//     PlcTask Inputs/GVL_iXlinker.EtherCAT_Master_BKCUCX.Beckhoff_CUxxxx.Beckhoff_CUxxxxEK1122.A_0001_CU1123_0000_0016.A_0002_CU1123_0010_0016.A_0003_CU1124_0000_0016.A_0004_CU1128_0000_0000.A_0005_CU1128_0000_0001.A_0006_CU1128_0000_0002.A_0013_CU2508_0000_0019.EPM_Inputs_Channel_1.Dropped_frames_tx <-> EPM Inputs Channel 1/Dropped frames tx
//     PlcTask Inputs/GVL_iXlinker.EtherCAT_Master_BKCUCX.Beckhoff_CUxxxx.Beckhoff_CUxxxxEK1122.A_0001_CU1123_0000_0016.A_0002_CU1123_0010_0016.A_0003_CU1124_0000_0016.A_0004_CU1128_0000_0000.A_0005_CU1128_0000_0001.A_0006_CU1128_0000_0002.A_0013_CU2508_0000_0019.EPM_Inputs_Channel_2.Dropped_frames_tx <-> EPM Inputs Channel 2/Dropped frames tx
//     PlcTask Inputs/GVL_iXlinker.EtherCAT_Master_BKCUCX.Beckhoff_CUxxxx.Beckhoff_CUxxxxEK1122.A_0001_CU1123_0000_0016.A_0002_CU1123_0010_0016.A_0003_CU1124_0000_0016.A_0004_CU1128_0000_0000.A_0005_CU1128_0000_0001.A_0006_CU1128_0000_0002.A_0013_CU2508_0000_0019.EPM_Inputs_Channel_3.Dropped_frames_tx <-> EPM Inputs Channel 3/Dropped frames tx
//     PlcTask Inputs/GVL_iXlinker.EtherCAT_Master_BKCUCX.Beckhoff_CUxxxx.Beckhoff_CUxxxxEK1122.A_0001_CU1123_0000_0016.A_0002_CU1123_0010_0016.A_0003_CU1124_0000_0016.A_0004_CU1128_0000_0000.A_0005_CU1128_0000_0001.A_0006_CU1128_0000_0002.A_0013_CU2508_0000_0019.EPM_Inputs_Channel_4.Dropped_frames_tx <-> EPM Inputs Channel 4/Dropped frames tx
//     PlcTask Inputs/GVL_iXlinker.EtherCAT_Master_BKCUCX.Beckhoff_CUxxxx.Beckhoff_CUxxxxEK1122.A_0001_CU1123_0000_0016.A_0002_CU1123_0010_0016.A_0003_CU1124_0000_0016.A_0004_CU1128_0000_0000.A_0005_CU1128_0000_0001.A_0006_CU1128_0000_0002.A_0013_CU2508_0000_0019.EPM_Inputs_Channel_5.Dropped_frames_tx <-> EPM Inputs Channel 5/Dropped frames tx
//     PlcTask Inputs/GVL_iXlinker.EtherCAT_Master_BKCUCX.Beckhoff_CUxxxx.Beckhoff_CUxxxxEK1122.A_0001_CU1123_0000_0016.A_0002_CU1123_0010_0016.A_0003_CU1124_0000_0016.A_0004_CU1128_0000_0000.A_0005_CU1128_0000_0001.A_0006_CU1128_0000_0002.A_0013_CU2508_0000_0019.EPM_Inputs_Channel_6.Dropped_frames_tx <-> EPM Inputs Channel 6/Dropped frames tx
//     PlcTask Inputs/GVL_iXlinker.EtherCAT_Master_BKCUCX.Beckhoff_CUxxxx.Beckhoff_CUxxxxEK1122.A_0001_CU1123_0000_0016.A_0002_CU1123_0010_0016.A_0003_CU1124_0000_0016.A_0004_CU1128_0000_0000.A_0005_CU1128_0000_0001.A_0006_CU1128_0000_0002.A_0013_CU2508_0000_0019.EPM_Inputs_Channel_7.Dropped_frames_tx <-> EPM Inputs Channel 7/Dropped frames tx
//     PlcTask Inputs/GVL_iXlinker.EtherCAT_Master_BKCUCX.Beckhoff_CUxxxx.Beckhoff_CUxxxxEK1122.A_0001_CU1123_0000_0016.A_0002_CU1123_0010_0016.A_0003_CU1124_0000_0016.A_0004_CU1128_0000_0000.A_0005_CU1128_0000_0001.A_0006_CU1128_0000_0002.A_0013_CU2508_0000_0019.EPM_Inputs_Channel_8.Dropped_frames_tx <-> EPM Inputs Channel 8/Dropped frames tx
//     PlcTask Inputs/GVL_iXlinker.EtherCAT_Master_BKCUCX.Beckhoff_CUxxxx.Beckhoff_CUxxxxEK1122.A_0001_CU1123_0000_0016.A_0002_CU1123_0010_0016.A_0003_CU1124_0000_0016.A_0004_CU1128_0000_0000.A_0005_CU1128_0000_0001.A_0006_CU1128_0000_0002.A_0013_CU2508_0000_0019.EPM_Inputs_Channel_9.Dropped_frames_tx <-> EPM Inputs Channel 9/Dropped frames tx
//     PlcTask Inputs/GVL_iXlinker.EtherCAT_Master_BKCUCX.Beckhoff_CUxxxx.Beckhoff_CUxxxxEK1122.A_0001_CU1123_0000_0016.A_0002_CU1123_0010_0016.A_0003_CU1124_0000_0016.A_0004_CU1128_0000_0000.A_0005_CU1128_0000_0001.A_0006_CU1128_0000_0002.A_0013_CU2508_0000_0019.EPM_Inputs_Channel_10.Dropped_frames_tx <-> EPM Inputs Channel 10/Dropped frames tx
//     PlcTask Inputs/GVL_iXlinker.EtherCAT_Master_BKCUCX.Beckhoff_CUxxxx.Beckhoff_CUxxxxEK1122.A_0001_CU1123_0000_0016.A_0002_CU1123_0010_0016.A_0003_CU1124_0000_0016.A_0004_CU1128_0000_0000.A_0005_CU1128_0000_0001.A_0006_CU1128_0000_0002.A_0013_CU2508_0000_0019.WcState.WcState <-> WcState/WcState
//     PlcTask Inputs/GVL_iXlinker.EtherCAT_Master_BKCUCX.Beckhoff_CUxxxx.Beckhoff_CUxxxxEK1122.A_0001_CU1123_0000_0016.A_0002_CU1123_0010_0016.A_0003_CU1124_0000_0016.A_0004_CU1128_0000_0000.A_0005_CU1128_0000_0001.A_0006_CU1128_0000_0002.A_0013_CU2508_0000_0019.WcState.InputToggle <-> WcState/InputToggle
//     PlcTask Inputs/GVL_iXlinker.EtherCAT_Master_BKCUCX.Beckhoff_CUxxxx.Beckhoff_CUxxxxEK1122.A_0001_CU1123_0000_0016.A_0002_CU1123_0010_0016.A_0003_CU1124_0000_0016.A_0004_CU1128_0000_0000.A_0005_CU1128_0000_0001.A_0006_CU1128_0000_0002.A_0013_CU2508_0000_0019.InfoData.AdsAddr <-> InfoData/AdsAddr
//     PlcTask Inputs/GVL_iXlinker.EtherCAT_Master_BKCUCX.Beckhoff_CUxxxx.Beckhoff_CUxxxxEK1122.A_0001_CU1123_0000_0016.A_0002_CU1123_0010_0016.A_0003_CU1124_0000_0016.A_0004_CU1128_0000_0000.A_0005_CU1128_0000_0001.A_0006_CU1128_0000_0002.A_0013_CU2508_0000_0019.InfoData.State <-> InfoData/State
//   PLC/PLC Instance <-> EtherCAT Master BKCUCX/Beckhoff CUxxxx/Beckhoff CUxxxxEK1122/A_0001(CU1123-0000-0016)/A_0002(CU1123-0010-0016)/A_0003(CU1124-0000-0016)/A_0004(CU1128-0000-0000)/A_0005(CU1128-0000-0001)/A_0006(CU1128-0000-0002)/A_0006(CU1128-0000-0002)_2 (CU1128-B)
//     PlcTask Inputs/GVL_iXlinker.EtherCAT_Master_BKCUCX.Beckhoff_CUxxxx.Beckhoff_CUxxxxEK1122.A_0001_CU1123_0000_0016.A_0002_CU1123_0010_0016.A_0003_CU1124_0000_0016.A_0004_CU1128_0000_0000.A_0005_CU1128_0000_0001.A_0006_CU1128_0000_0002.A_0006_CU1128_0000_0002_2_CU1128_B.InfoData.State <-> InfoData/State
//   PLC/PLC Instance <-> EtherCAT Master BKCUCX/Beckhoff CUxxxx/Beckhoff CUxxxxEK1122/A_0001(CU1123-0000-0016)/A_0002(CU1123-0010-0016)/A_0003(CU1124-0000-0016)/A_0004(CU1128-0000-0000)/A_0005(CU1128-0000-0001)/A_0006(CU1128-0000-0002)/A_0006(CU1128-0000-0002)_3 (CU1128-C)
//     PlcTask Inputs/GVL_iXlinker.EtherCAT_Master_BKCUCX.Beckhoff_CUxxxx.Beckhoff_CUxxxxEK1122.A_0001_CU1123_0000_0016.A_0002_CU1123_0010_0016.A_0003_CU1124_0000_0016.A_0004_CU1128_0000_0000.A_0005_CU1128_0000_0001.A_0006_CU1128_0000_0002.A_0006_CU1128_0000_0002_3_CU1128_C.InfoData.State <-> InfoData/State
//   PLC/PLC Instance <-> EtherCAT Master BKCUCX/Beckhoff CUxxxx/Beckhoff CUxxxxEK1122/A_0001(CU1123-0000-0016)/A_0002(CU1123-0010-0016)/A_0003(CU1124-0000-0016)/A_0004(CU1128-0000-0000)/A_0005(CU1128-0000-0001)/A_0005(CU1128-0000-0001)_2 (CU1128-B)
//     PlcTask Inputs/GVL_iXlinker.EtherCAT_Master_BKCUCX.Beckhoff_CUxxxx.Beckhoff_CUxxxxEK1122.A_0001_CU1123_0000_0016.A_0002_CU1123_0010_0016.A_0003_CU1124_0000_0016.A_0004_CU1128_0000_0000.A_0005_CU1128_0000_0001.A_0005_CU1128_0000_0001_2_CU1128_B.InfoData.State <-> InfoData/State
//   PLC/PLC Instance <-> EtherCAT Master BKCUCX/Beckhoff CUxxxx/Beckhoff CUxxxxEK1122/A_0001(CU1123-0000-0016)/A_0002(CU1123-0010-0016)/A_0003(CU1124-0000-0016)/A_0004(CU1128-0000-0000)/A_0005(CU1128-0000-0001)/A_0005(CU1128-0000-0001)_3 (CU1128-C)
//     PlcTask Inputs/GVL_iXlinker.EtherCAT_Master_BKCUCX.Beckhoff_CUxxxx.Beckhoff_CUxxxxEK1122.A_0001_CU1123_0000_0016.A_0002_CU1123_0010_0016.A_0003_CU1124_0000_0016.A_0004_CU1128_0000_0000.A_0005_CU1128_0000_0001.A_0005_CU1128_0000_0001_3_CU1128_C.InfoData.State <-> InfoData/State
//   PLC/PLC Instance <-> EtherCAT Master BKCUCX/Beckhoff CUxxxx/Beckhoff CUxxxxEK1122/A_0001(CU1123-0000-0016)/A_0002(CU1123-0010-0016)/A_0003(CU1124-0000-0016)/A_0004(CU1128-0000-0000)/A_0004(CU1128-0000-0000)_2 (CU1128-B)
//     PlcTask Inputs/GVL_iXlinker.EtherCAT_Master_BKCUCX.Beckhoff_CUxxxx.Beckhoff_CUxxxxEK1122.A_0001_CU1123_0000_0016.A_0002_CU1123_0010_0016.A_0003_CU1124_0000_0016.A_0004_CU1128_0000_0000.A_0004_CU1128_0000_0000_2_CU1128_B.InfoData.State <-> InfoData/State
//   PLC/PLC Instance <-> EtherCAT Master BKCUCX/Beckhoff CUxxxx/Beckhoff CUxxxxEK1122/A_0001(CU1123-0000-0016)/A_0002(CU1123-0010-0016)/A_0003(CU1124-0000-0016)/A_0004(CU1128-0000-0000)/A_0004(CU1128-0000-0000)_3 (CU1128-C)
//     PlcTask Inputs/GVL_iXlinker.EtherCAT_Master_BKCUCX.Beckhoff_CUxxxx.Beckhoff_CUxxxxEK1122.A_0001_CU1123_0000_0016.A_0002_CU1123_0010_0016.A_0003_CU1124_0000_0016.A_0004_CU1128_0000_0000.A_0004_CU1128_0000_0000_3_CU1128_C.InfoData.State <-> InfoData/State
//   PLC/PLC Instance <-> EtherCAT Master BKCUCX/Beckhoff CXxxxx
//     PlcTask Inputs/GVL_iXlinker.EtherCAT_Master_BKCUCX.Beckhoff_CXxxxx.InfoData.State <-> InfoData/State
//   PLC/PLC Instance <-> EtherCAT Master BKCUCX/Beckhoff CXxxxx/Beckhoff CXxxxxEK1122
//     PlcTask Inputs/GVL_iXlinker.EtherCAT_Master_BKCUCX.Beckhoff_CXxxxx.Beckhoff_CXxxxxEK1122.InfoData.State <-> InfoData/State
//   PLC/PLC Instance <-> EtherCAT Master BKCUCX/Beckhoff CXxxxx/Beckhoff CXxxxxEK1122/Beckhoff CXxxxxsub EK1100
//     PlcTask Inputs/GVL_iXlinker.EtherCAT_Master_BKCUCX.Beckhoff_CXxxxx.Beckhoff_CXxxxxEK1122.Beckhoff_CXxxxxsub_EK1100.InfoData.State <-> InfoData/State
//   PLC/PLC Instance <-> EtherCAT Master BKCUCX/Beckhoff CXxxxx/Beckhoff CXxxxxEK1122/A_0001(CX1100-0004-0000)
//     PlcTask Inputs/GVL_iXlinker.EtherCAT_Master_BKCUCX.Beckhoff_CXxxxx.Beckhoff_CXxxxxEK1122.A_0001_CX1100_0004_0000.InfoData.State <-> InfoData/State
//   PLC/PLC Instance <-> EtherCAT Master BKCUCX/Beckhoff CXxxxx/Beckhoff CXxxxxEK1122/A_0003(CX1100-0004-0002)
//     PlcTask Inputs/GVL_iXlinker.EtherCAT_Master_BKCUCX.Beckhoff_CXxxxx.Beckhoff_CXxxxxEK1122.A_0003_CX1100_0004_0002.InfoData.State <-> InfoData/State
//   PLC/PLC Instance <-> EtherCAT Master BKCUCX/Beckhoff CXxxxx/Beckhoff CXxxxxEK1122/A_0004 (CX5010 EtherCAT slave)
//     PlcTask Inputs/GVL_iXlinker.EtherCAT_Master_BKCUCX.Beckhoff_CXxxxx.Beckhoff_CXxxxxEK1122.A_0004_CX5010_EtherCAT_slave.Device_Status_Mapping.TxPdoState <-> Device Status Mapping/TxPdoState
//     PlcTask Inputs/GVL_iXlinker.EtherCAT_Master_BKCUCX.Beckhoff_CXxxxx.Beckhoff_CXxxxxEK1122.A_0004_CX5010_EtherCAT_slave.Device_Status_Mapping.TxPdoToggle <-> Device Status Mapping/TxPdoToggle
//     PlcTask Inputs/GVL_iXlinker.EtherCAT_Master_BKCUCX.Beckhoff_CXxxxx.Beckhoff_CXxxxxEK1122.A_0004_CX5010_EtherCAT_slave.WcState.WcState <-> WcState/WcState
//     PlcTask Inputs/GVL_iXlinker.EtherCAT_Master_BKCUCX.Beckhoff_CXxxxx.Beckhoff_CXxxxxEK1122.A_0004_CX5010_EtherCAT_slave.WcState.InputToggle <-> WcState/InputToggle
//     PlcTask Inputs/GVL_iXlinker.EtherCAT_Master_BKCUCX.Beckhoff_CXxxxx.Beckhoff_CXxxxxEK1122.A_0004_CX5010_EtherCAT_slave.InfoData.AdsAddr <-> InfoData/AdsAddr
//     PlcTask Inputs/GVL_iXlinker.EtherCAT_Master_BKCUCX.Beckhoff_CXxxxx.Beckhoff_CXxxxxEK1122.A_0004_CX5010_EtherCAT_slave.InfoData.AoeNetId <-> InfoData/AoeNetId
//     PlcTask Inputs/GVL_iXlinker.EtherCAT_Master_BKCUCX.Beckhoff_CXxxxx.Beckhoff_CXxxxxEK1122.A_0004_CX5010_EtherCAT_slave.InfoData.State <-> InfoData/State
//   PLC/PLC Instance <-> EtherCAT Master BKCUCX/Beckhoff CXxxxx/Beckhoff CXxxxxEK1122/A_0005 (CX5010 EtherCAT slave)
//     PlcTask Inputs/GVL_iXlinker.EtherCAT_Master_BKCUCX.Beckhoff_CXxxxx.Beckhoff_CXxxxxEK1122.A_0005_CX5010_EtherCAT_slave.Device_Status_Mapping.TxPdoState <-> Device Status Mapping/TxPdoState
//     PlcTask Inputs/GVL_iXlinker.EtherCAT_Master_BKCUCX.Beckhoff_CXxxxx.Beckhoff_CXxxxxEK1122.A_0005_CX5010_EtherCAT_slave.Device_Status_Mapping.TxPdoToggle <-> Device Status Mapping/TxPdoToggle
//     PlcTask Inputs/GVL_iXlinker.EtherCAT_Master_BKCUCX.Beckhoff_CXxxxx.Beckhoff_CXxxxxEK1122.A_0005_CX5010_EtherCAT_slave.WcState.WcState <-> WcState/WcState
//     PlcTask Inputs/GVL_iXlinker.EtherCAT_Master_BKCUCX.Beckhoff_CXxxxx.Beckhoff_CXxxxxEK1122.A_0005_CX5010_EtherCAT_slave.WcState.InputToggle <-> WcState/InputToggle
//     PlcTask Inputs/GVL_iXlinker.EtherCAT_Master_BKCUCX.Beckhoff_CXxxxx.Beckhoff_CXxxxxEK1122.A_0005_CX5010_EtherCAT_slave.InfoData.AdsAddr <-> InfoData/AdsAddr
//     PlcTask Inputs/GVL_iXlinker.EtherCAT_Master_BKCUCX.Beckhoff_CXxxxx.Beckhoff_CXxxxxEK1122.A_0005_CX5010_EtherCAT_slave.InfoData.AoeNetId <-> InfoData/AoeNetId
//     PlcTask Inputs/GVL_iXlinker.EtherCAT_Master_BKCUCX.Beckhoff_CXxxxx.Beckhoff_CXxxxxEK1122.A_0005_CX5010_EtherCAT_slave.InfoData.State <-> InfoData/State
//   PLC/PLC Instance <-> EtherCAT Master BKCUCX/Beckhoff CXxxxx/Beckhoff CXxxxxEK1122/A_0006 (CX5020 EtherCAT slave)
//     PlcTask Inputs/GVL_iXlinker.EtherCAT_Master_BKCUCX.Beckhoff_CXxxxx.Beckhoff_CXxxxxEK1122.A_0006_CX5020_EtherCAT_slave.Device_Status_Mapping.TxPdoState <-> Device Status Mapping/TxPdoState
//     PlcTask Inputs/GVL_iXlinker.EtherCAT_Master_BKCUCX.Beckhoff_CXxxxx.Beckhoff_CXxxxxEK1122.A_0006_CX5020_EtherCAT_slave.Device_Status_Mapping.TxPdoToggle <-> Device Status Mapping/TxPdoToggle
//     PlcTask Inputs/GVL_iXlinker.EtherCAT_Master_BKCUCX.Beckhoff_CXxxxx.Beckhoff_CXxxxxEK1122.A_0006_CX5020_EtherCAT_slave.WcState.WcState <-> WcState/WcState
//     PlcTask Inputs/GVL_iXlinker.EtherCAT_Master_BKCUCX.Beckhoff_CXxxxx.Beckhoff_CXxxxxEK1122.A_0006_CX5020_EtherCAT_slave.WcState.InputToggle <-> WcState/InputToggle
//     PlcTask Inputs/GVL_iXlinker.EtherCAT_Master_BKCUCX.Beckhoff_CXxxxx.Beckhoff_CXxxxxEK1122.A_0006_CX5020_EtherCAT_slave.InfoData.AdsAddr <-> InfoData/AdsAddr
//     PlcTask Inputs/GVL_iXlinker.EtherCAT_Master_BKCUCX.Beckhoff_CXxxxx.Beckhoff_CXxxxxEK1122.A_0006_CX5020_EtherCAT_slave.InfoData.AoeNetId <-> InfoData/AoeNetId
//     PlcTask Inputs/GVL_iXlinker.EtherCAT_Master_BKCUCX.Beckhoff_CXxxxx.Beckhoff_CXxxxxEK1122.A_0006_CX5020_EtherCAT_slave.InfoData.State <-> InfoData/State
//   PLC/PLC Instance <-> EtherCAT Master BKCUCX/Beckhoff CXxxxx/Beckhoff CXxxxxEK1122/A_0007 (CX5020 EtherCAT slave)
//     PlcTask Inputs/GVL_iXlinker.EtherCAT_Master_BKCUCX.Beckhoff_CXxxxx.Beckhoff_CXxxxxEK1122.A_0007_CX5020_EtherCAT_slave.Device_Status_Mapping.TxPdoState <-> Device Status Mapping/TxPdoState
//     PlcTask Inputs/GVL_iXlinker.EtherCAT_Master_BKCUCX.Beckhoff_CXxxxx.Beckhoff_CXxxxxEK1122.A_0007_CX5020_EtherCAT_slave.Device_Status_Mapping.TxPdoToggle <-> Device Status Mapping/TxPdoToggle
//     PlcTask Inputs/GVL_iXlinker.EtherCAT_Master_BKCUCX.Beckhoff_CXxxxx.Beckhoff_CXxxxxEK1122.A_0007_CX5020_EtherCAT_slave.WcState.WcState <-> WcState/WcState
//     PlcTask Inputs/GVL_iXlinker.EtherCAT_Master_BKCUCX.Beckhoff_CXxxxx.Beckhoff_CXxxxxEK1122.A_0007_CX5020_EtherCAT_slave.WcState.InputToggle <-> WcState/InputToggle
//     PlcTask Inputs/GVL_iXlinker.EtherCAT_Master_BKCUCX.Beckhoff_CXxxxx.Beckhoff_CXxxxxEK1122.A_0007_CX5020_EtherCAT_slave.InfoData.AdsAddr <-> InfoData/AdsAddr
//     PlcTask Inputs/GVL_iXlinker.EtherCAT_Master_BKCUCX.Beckhoff_CXxxxx.Beckhoff_CXxxxxEK1122.A_0007_CX5020_EtherCAT_slave.InfoData.AoeNetId <-> InfoData/AoeNetId
//     PlcTask Inputs/GVL_iXlinker.EtherCAT_Master_BKCUCX.Beckhoff_CXxxxx.Beckhoff_CXxxxxEK1122.A_0007_CX5020_EtherCAT_slave.InfoData.State <-> InfoData/State
//   PLC/PLC Instance <-> EtherCAT Master BKCUCX/Beckhoff CXxxxx/Beckhoff CXxxxxEK1122/A_0008 (CX8010 EtherCAT slave)
//     PlcTask Inputs/GVL_iXlinker.EtherCAT_Master_BKCUCX.Beckhoff_CXxxxx.Beckhoff_CXxxxxEK1122.A_0008_CX8010_EtherCAT_slave.Device_Status_Mapping.TxPdoState <-> Device Status Mapping/TxPdoState
//     PlcTask Inputs/GVL_iXlinker.EtherCAT_Master_BKCUCX.Beckhoff_CXxxxx.Beckhoff_CXxxxxEK1122.A_0008_CX8010_EtherCAT_slave.Device_Status_Mapping.TxPdoToggle <-> Device Status Mapping/TxPdoToggle
//     PlcTask Inputs/GVL_iXlinker.EtherCAT_Master_BKCUCX.Beckhoff_CXxxxx.Beckhoff_CXxxxxEK1122.A_0008_CX8010_EtherCAT_slave.WcState.WcState <-> WcState/WcState
//     PlcTask Inputs/GVL_iXlinker.EtherCAT_Master_BKCUCX.Beckhoff_CXxxxx.Beckhoff_CXxxxxEK1122.A_0008_CX8010_EtherCAT_slave.WcState.InputToggle <-> WcState/InputToggle
//     PlcTask Inputs/GVL_iXlinker.EtherCAT_Master_BKCUCX.Beckhoff_CXxxxx.Beckhoff_CXxxxxEK1122.A_0008_CX8010_EtherCAT_slave.InfoData.AdsAddr <-> InfoData/AdsAddr
//     PlcTask Inputs/GVL_iXlinker.EtherCAT_Master_BKCUCX.Beckhoff_CXxxxx.Beckhoff_CXxxxxEK1122.A_0008_CX8010_EtherCAT_slave.InfoData.AoeNetId <-> InfoData/AoeNetId
//     PlcTask Inputs/GVL_iXlinker.EtherCAT_Master_BKCUCX.Beckhoff_CXxxxx.Beckhoff_CXxxxxEK1122.A_0008_CX8010_EtherCAT_slave.InfoData.State <-> InfoData/State
//   PLC/PLC Instance <-> EtherCAT Master BKCUCX/Beckhoff CXxxxx/Beckhoff CXxxxxEK1122/A_0009 (CX8010 EtherCAT slave)
//     PlcTask Inputs/GVL_iXlinker.EtherCAT_Master_BKCUCX.Beckhoff_CXxxxx.Beckhoff_CXxxxxEK1122.A_0009_CX8010_EtherCAT_slave.Device_Status_Mapping.TxPdoState <-> Device Status Mapping/TxPdoState
//     PlcTask Inputs/GVL_iXlinker.EtherCAT_Master_BKCUCX.Beckhoff_CXxxxx.Beckhoff_CXxxxxEK1122.A_0009_CX8010_EtherCAT_slave.Device_Status_Mapping.TxPdoToggle <-> Device Status Mapping/TxPdoToggle
//     PlcTask Inputs/GVL_iXlinker.EtherCAT_Master_BKCUCX.Beckhoff_CXxxxx.Beckhoff_CXxxxxEK1122.A_0009_CX8010_EtherCAT_slave.WcState.WcState <-> WcState/WcState
//     PlcTask Inputs/GVL_iXlinker.EtherCAT_Master_BKCUCX.Beckhoff_CXxxxx.Beckhoff_CXxxxxEK1122.A_0009_CX8010_EtherCAT_slave.WcState.InputToggle <-> WcState/InputToggle
//     PlcTask Inputs/GVL_iXlinker.EtherCAT_Master_BKCUCX.Beckhoff_CXxxxx.Beckhoff_CXxxxxEK1122.A_0009_CX8010_EtherCAT_slave.InfoData.AdsAddr <-> InfoData/AdsAddr
//     PlcTask Inputs/GVL_iXlinker.EtherCAT_Master_BKCUCX.Beckhoff_CXxxxx.Beckhoff_CXxxxxEK1122.A_0009_CX8010_EtherCAT_slave.InfoData.AoeNetId <-> InfoData/AoeNetId
//     PlcTask Inputs/GVL_iXlinker.EtherCAT_Master_BKCUCX.Beckhoff_CXxxxx.Beckhoff_CXxxxxEK1122.A_0009_CX8010_EtherCAT_slave.InfoData.State <-> InfoData/State
//   PLC/PLC Instance <-> EtherCAT Master BKCUCX/Beckhoff CXxxxx/Beckhoff CXxxxxEK1122/A_0010 (CX8110 EtherCAT slave)
//     PlcTask Inputs/GVL_iXlinker.EtherCAT_Master_BKCUCX.Beckhoff_CXxxxx.Beckhoff_CXxxxxEK1122.A_0010_CX8110_EtherCAT_slave.Device_Status_Mapping.TxPdoState <-> Device Status Mapping/TxPdoState
//     PlcTask Inputs/GVL_iXlinker.EtherCAT_Master_BKCUCX.Beckhoff_CXxxxx.Beckhoff_CXxxxxEK1122.A_0010_CX8110_EtherCAT_slave.Device_Status_Mapping.TxPdoToggle <-> Device Status Mapping/TxPdoToggle
//     PlcTask Inputs/GVL_iXlinker.EtherCAT_Master_BKCUCX.Beckhoff_CXxxxx.Beckhoff_CXxxxxEK1122.A_0010_CX8110_EtherCAT_slave.WcState.WcState <-> WcState/WcState
//     PlcTask Inputs/GVL_iXlinker.EtherCAT_Master_BKCUCX.Beckhoff_CXxxxx.Beckhoff_CXxxxxEK1122.A_0010_CX8110_EtherCAT_slave.WcState.InputToggle <-> WcState/InputToggle
//     PlcTask Inputs/GVL_iXlinker.EtherCAT_Master_BKCUCX.Beckhoff_CXxxxx.Beckhoff_CXxxxxEK1122.A_0010_CX8110_EtherCAT_slave.InfoData.AdsAddr <-> InfoData/AdsAddr
//     PlcTask Inputs/GVL_iXlinker.EtherCAT_Master_BKCUCX.Beckhoff_CXxxxx.Beckhoff_CXxxxxEK1122.A_0010_CX8110_EtherCAT_slave.InfoData.AoeNetId <-> InfoData/AoeNetId
//     PlcTask Inputs/GVL_iXlinker.EtherCAT_Master_BKCUCX.Beckhoff_CXxxxx.Beckhoff_CXxxxxEK1122.A_0010_CX8110_EtherCAT_slave.InfoData.State <-> InfoData/State
//   PLC/PLC Instance <-> EtherCAT Master BKCUCX/Beckhoff CXxxxx/Beckhoff CXxxxxEK1122/A_0011 (CX2020 EtherCAT slave)
//     PlcTask Inputs/GVL_iXlinker.EtherCAT_Master_BKCUCX.Beckhoff_CXxxxx.Beckhoff_CXxxxxEK1122.A_0011_CX2020_EtherCAT_slave.Device_Status_Mapping.TxPdoState <-> Device Status Mapping/TxPdoState
//     PlcTask Inputs/GVL_iXlinker.EtherCAT_Master_BKCUCX.Beckhoff_CXxxxx.Beckhoff_CXxxxxEK1122.A_0011_CX2020_EtherCAT_slave.Device_Status_Mapping.TxPdoToggle <-> Device Status Mapping/TxPdoToggle
//     PlcTask Inputs/GVL_iXlinker.EtherCAT_Master_BKCUCX.Beckhoff_CXxxxx.Beckhoff_CXxxxxEK1122.A_0011_CX2020_EtherCAT_slave.WcState.WcState <-> WcState/WcState
//     PlcTask Inputs/GVL_iXlinker.EtherCAT_Master_BKCUCX.Beckhoff_CXxxxx.Beckhoff_CXxxxxEK1122.A_0011_CX2020_EtherCAT_slave.WcState.InputToggle <-> WcState/InputToggle
//     PlcTask Inputs/GVL_iXlinker.EtherCAT_Master_BKCUCX.Beckhoff_CXxxxx.Beckhoff_CXxxxxEK1122.A_0011_CX2020_EtherCAT_slave.InfoData.AdsAddr <-> InfoData/AdsAddr
//     PlcTask Inputs/GVL_iXlinker.EtherCAT_Master_BKCUCX.Beckhoff_CXxxxx.Beckhoff_CXxxxxEK1122.A_0011_CX2020_EtherCAT_slave.InfoData.AoeNetId <-> InfoData/AoeNetId
//     PlcTask Inputs/GVL_iXlinker.EtherCAT_Master_BKCUCX.Beckhoff_CXxxxx.Beckhoff_CXxxxxEK1122.A_0011_CX2020_EtherCAT_slave.InfoData.State <-> InfoData/State
//   PLC/PLC Instance <-> EtherCAT Master BKCUCX/Beckhoff CXxxxx/Beckhoff CXxxxxEK1122/A_0012 (CX2020 EtherCAT slave)
//     PlcTask Inputs/GVL_iXlinker.EtherCAT_Master_BKCUCX.Beckhoff_CXxxxx.Beckhoff_CXxxxxEK1122.A_0012_CX2020_EtherCAT_slave.Device_Status_Mapping.TxPdoState <-> Device Status Mapping/TxPdoState
//     PlcTask Inputs/GVL_iXlinker.EtherCAT_Master_BKCUCX.Beckhoff_CXxxxx.Beckhoff_CXxxxxEK1122.A_0012_CX2020_EtherCAT_slave.Device_Status_Mapping.TxPdoToggle <-> Device Status Mapping/TxPdoToggle
//     PlcTask Inputs/GVL_iXlinker.EtherCAT_Master_BKCUCX.Beckhoff_CXxxxx.Beckhoff_CXxxxxEK1122.A_0012_CX2020_EtherCAT_slave.WcState.WcState <-> WcState/WcState
//     PlcTask Inputs/GVL_iXlinker.EtherCAT_Master_BKCUCX.Beckhoff_CXxxxx.Beckhoff_CXxxxxEK1122.A_0012_CX2020_EtherCAT_slave.WcState.InputToggle <-> WcState/InputToggle
//     PlcTask Inputs/GVL_iXlinker.EtherCAT_Master_BKCUCX.Beckhoff_CXxxxx.Beckhoff_CXxxxxEK1122.A_0012_CX2020_EtherCAT_slave.InfoData.AdsAddr <-> InfoData/AdsAddr
//     PlcTask Inputs/GVL_iXlinker.EtherCAT_Master_BKCUCX.Beckhoff_CXxxxx.Beckhoff_CXxxxxEK1122.A_0012_CX2020_EtherCAT_slave.InfoData.AoeNetId <-> InfoData/AoeNetId
//     PlcTask Inputs/GVL_iXlinker.EtherCAT_Master_BKCUCX.Beckhoff_CXxxxx.Beckhoff_CXxxxxEK1122.A_0012_CX2020_EtherCAT_slave.InfoData.State <-> InfoData/State
//   PLC/PLC Instance <-> EtherCAT Master BKCUCX/Beckhoff CXxxxx/Beckhoff CXxxxxEK1122/A_0013 (CX2020 EtherCAT slave)
//     PlcTask Inputs/GVL_iXlinker.EtherCAT_Master_BKCUCX.Beckhoff_CXxxxx.Beckhoff_CXxxxxEK1122.A_0013_CX2020_EtherCAT_slave.Device_Status_Mapping.TxPdoState <-> Device Status Mapping/TxPdoState
//     PlcTask Inputs/GVL_iXlinker.EtherCAT_Master_BKCUCX.Beckhoff_CXxxxx.Beckhoff_CXxxxxEK1122.A_0013_CX2020_EtherCAT_slave.Device_Status_Mapping.TxPdoToggle <-> Device Status Mapping/TxPdoToggle
//     PlcTask Inputs/GVL_iXlinker.EtherCAT_Master_BKCUCX.Beckhoff_CXxxxx.Beckhoff_CXxxxxEK1122.A_0013_CX2020_EtherCAT_slave.WcState.WcState <-> WcState/WcState
//     PlcTask Inputs/GVL_iXlinker.EtherCAT_Master_BKCUCX.Beckhoff_CXxxxx.Beckhoff_CXxxxxEK1122.A_0013_CX2020_EtherCAT_slave.WcState.InputToggle <-> WcState/InputToggle
//     PlcTask Inputs/GVL_iXlinker.EtherCAT_Master_BKCUCX.Beckhoff_CXxxxx.Beckhoff_CXxxxxEK1122.A_0013_CX2020_EtherCAT_slave.InfoData.AdsAddr <-> InfoData/AdsAddr
//     PlcTask Inputs/GVL_iXlinker.EtherCAT_Master_BKCUCX.Beckhoff_CXxxxx.Beckhoff_CXxxxxEK1122.A_0013_CX2020_EtherCAT_slave.InfoData.AoeNetId <-> InfoData/AoeNetId
//     PlcTask Inputs/GVL_iXlinker.EtherCAT_Master_BKCUCX.Beckhoff_CXxxxx.Beckhoff_CXxxxxEK1122.A_0013_CX2020_EtherCAT_slave.InfoData.State <-> InfoData/State
//   PLC/PLC Instance <-> EtherCAT Master BKCUCX/Beckhoff CXxxxx/Beckhoff CXxxxxEK1122/A_0014 (CX2030 EtherCAT slave)
//     PlcTask Inputs/GVL_iXlinker.EtherCAT_Master_BKCUCX.Beckhoff_CXxxxx.Beckhoff_CXxxxxEK1122.A_0014_CX2030_EtherCAT_slave.Device_Status_Mapping.TxPdoState <-> Device Status Mapping/TxPdoState
//     PlcTask Inputs/GVL_iXlinker.EtherCAT_Master_BKCUCX.Beckhoff_CXxxxx.Beckhoff_CXxxxxEK1122.A_0014_CX2030_EtherCAT_slave.Device_Status_Mapping.TxPdoToggle <-> Device Status Mapping/TxPdoToggle
//     PlcTask Inputs/GVL_iXlinker.EtherCAT_Master_BKCUCX.Beckhoff_CXxxxx.Beckhoff_CXxxxxEK1122.A_0014_CX2030_EtherCAT_slave.WcState.WcState <-> WcState/WcState
//     PlcTask Inputs/GVL_iXlinker.EtherCAT_Master_BKCUCX.Beckhoff_CXxxxx.Beckhoff_CXxxxxEK1122.A_0014_CX2030_EtherCAT_slave.WcState.InputToggle <-> WcState/InputToggle
//     PlcTask Inputs/GVL_iXlinker.EtherCAT_Master_BKCUCX.Beckhoff_CXxxxx.Beckhoff_CXxxxxEK1122.A_0014_CX2030_EtherCAT_slave.InfoData.AdsAddr <-> InfoData/AdsAddr
//     PlcTask Inputs/GVL_iXlinker.EtherCAT_Master_BKCUCX.Beckhoff_CXxxxx.Beckhoff_CXxxxxEK1122.A_0014_CX2030_EtherCAT_slave.InfoData.AoeNetId <-> InfoData/AoeNetId
//     PlcTask Inputs/GVL_iXlinker.EtherCAT_Master_BKCUCX.Beckhoff_CXxxxx.Beckhoff_CXxxxxEK1122.A_0014_CX2030_EtherCAT_slave.InfoData.State <-> InfoData/State
//   PLC/PLC Instance <-> EtherCAT Master BKCUCX/Beckhoff CXxxxx/Beckhoff CXxxxxEK1122/A_0015 (CX2030 EtherCAT slave)
//     PlcTask Inputs/GVL_iXlinker.EtherCAT_Master_BKCUCX.Beckhoff_CXxxxx.Beckhoff_CXxxxxEK1122.A_0015_CX2030_EtherCAT_slave.Device_Status_Mapping.TxPdoState <-> Device Status Mapping/TxPdoState
//     PlcTask Inputs/GVL_iXlinker.EtherCAT_Master_BKCUCX.Beckhoff_CXxxxx.Beckhoff_CXxxxxEK1122.A_0015_CX2030_EtherCAT_slave.Device_Status_Mapping.TxPdoToggle <-> Device Status Mapping/TxPdoToggle
//     PlcTask Inputs/GVL_iXlinker.EtherCAT_Master_BKCUCX.Beckhoff_CXxxxx.Beckhoff_CXxxxxEK1122.A_0015_CX2030_EtherCAT_slave.WcState.WcState <-> WcState/WcState
//     PlcTask Inputs/GVL_iXlinker.EtherCAT_Master_BKCUCX.Beckhoff_CXxxxx.Beckhoff_CXxxxxEK1122.A_0015_CX2030_EtherCAT_slave.WcState.InputToggle <-> WcState/InputToggle
//     PlcTask Inputs/GVL_iXlinker.EtherCAT_Master_BKCUCX.Beckhoff_CXxxxx.Beckhoff_CXxxxxEK1122.A_0015_CX2030_EtherCAT_slave.InfoData.AdsAddr <-> InfoData/AdsAddr
//     PlcTask Inputs/GVL_iXlinker.EtherCAT_Master_BKCUCX.Beckhoff_CXxxxx.Beckhoff_CXxxxxEK1122.A_0015_CX2030_EtherCAT_slave.InfoData.AoeNetId <-> InfoData/AoeNetId
//     PlcTask Inputs/GVL_iXlinker.EtherCAT_Master_BKCUCX.Beckhoff_CXxxxx.Beckhoff_CXxxxxEK1122.A_0015_CX2030_EtherCAT_slave.InfoData.State <-> InfoData/State
//   PLC/PLC Instance <-> EtherCAT Master BKCUCX/Beckhoff CXxxxx/Beckhoff CXxxxxEK1122/A_0016 (CX2030 EtherCAT slave)
//     PlcTask Inputs/GVL_iXlinker.EtherCAT_Master_BKCUCX.Beckhoff_CXxxxx.Beckhoff_CXxxxxEK1122.A_0016_CX2030_EtherCAT_slave.Device_Status_Mapping.TxPdoState <-> Device Status Mapping/TxPdoState
//     PlcTask Inputs/GVL_iXlinker.EtherCAT_Master_BKCUCX.Beckhoff_CXxxxx.Beckhoff_CXxxxxEK1122.A_0016_CX2030_EtherCAT_slave.Device_Status_Mapping.TxPdoToggle <-> Device Status Mapping/TxPdoToggle
//     PlcTask Inputs/GVL_iXlinker.EtherCAT_Master_BKCUCX.Beckhoff_CXxxxx.Beckhoff_CXxxxxEK1122.A_0016_CX2030_EtherCAT_slave.WcState.WcState <-> WcState/WcState
//     PlcTask Inputs/GVL_iXlinker.EtherCAT_Master_BKCUCX.Beckhoff_CXxxxx.Beckhoff_CXxxxxEK1122.A_0016_CX2030_EtherCAT_slave.WcState.InputToggle <-> WcState/InputToggle
//     PlcTask Inputs/GVL_iXlinker.EtherCAT_Master_BKCUCX.Beckhoff_CXxxxx.Beckhoff_CXxxxxEK1122.A_0016_CX2030_EtherCAT_slave.InfoData.AdsAddr <-> InfoData/AdsAddr
//     PlcTask Inputs/GVL_iXlinker.EtherCAT_Master_BKCUCX.Beckhoff_CXxxxx.Beckhoff_CXxxxxEK1122.A_0016_CX2030_EtherCAT_slave.InfoData.AoeNetId <-> InfoData/AoeNetId
//     PlcTask Inputs/GVL_iXlinker.EtherCAT_Master_BKCUCX.Beckhoff_CXxxxx.Beckhoff_CXxxxxEK1122.A_0016_CX2030_EtherCAT_slave.InfoData.State <-> InfoData/State
//   PLC/PLC Instance <-> EtherCAT Master BKCUCX/Beckhoff CXxxxx/Beckhoff CXxxxxEK1122/A_0017 (CX2033 EtherCAT slave)
//     PlcTask Inputs/GVL_iXlinker.EtherCAT_Master_BKCUCX.Beckhoff_CXxxxx.Beckhoff_CXxxxxEK1122.A_0017_CX2033_EtherCAT_slave.Device_Status_Mapping.TxPdoState <-> Device Status Mapping/TxPdoState
//     PlcTask Inputs/GVL_iXlinker.EtherCAT_Master_BKCUCX.Beckhoff_CXxxxx.Beckhoff_CXxxxxEK1122.A_0017_CX2033_EtherCAT_slave.Device_Status_Mapping.TxPdoToggle <-> Device Status Mapping/TxPdoToggle
//     PlcTask Inputs/GVL_iXlinker.EtherCAT_Master_BKCUCX.Beckhoff_CXxxxx.Beckhoff_CXxxxxEK1122.A_0017_CX2033_EtherCAT_slave.WcState.WcState <-> WcState/WcState
//     PlcTask Inputs/GVL_iXlinker.EtherCAT_Master_BKCUCX.Beckhoff_CXxxxx.Beckhoff_CXxxxxEK1122.A_0017_CX2033_EtherCAT_slave.WcState.InputToggle <-> WcState/InputToggle
//     PlcTask Inputs/GVL_iXlinker.EtherCAT_Master_BKCUCX.Beckhoff_CXxxxx.Beckhoff_CXxxxxEK1122.A_0017_CX2033_EtherCAT_slave.InfoData.AdsAddr <-> InfoData/AdsAddr
//     PlcTask Inputs/GVL_iXlinker.EtherCAT_Master_BKCUCX.Beckhoff_CXxxxx.Beckhoff_CXxxxxEK1122.A_0017_CX2033_EtherCAT_slave.InfoData.AoeNetId <-> InfoData/AoeNetId
//     PlcTask Inputs/GVL_iXlinker.EtherCAT_Master_BKCUCX.Beckhoff_CXxxxx.Beckhoff_CXxxxxEK1122.A_0017_CX2033_EtherCAT_slave.InfoData.State <-> InfoData/State
//   PLC/PLC Instance <-> EtherCAT Master BKCUCX/Beckhoff CXxxxx/Beckhoff CXxxxxEK1122/A_0018 (CX2040 EtherCAT slave)
//     PlcTask Inputs/GVL_iXlinker.EtherCAT_Master_BKCUCX.Beckhoff_CXxxxx.Beckhoff_CXxxxxEK1122.A_0018_CX2040_EtherCAT_slave.Device_Status_Mapping.TxPdoState <-> Device Status Mapping/TxPdoState
//     PlcTask Inputs/GVL_iXlinker.EtherCAT_Master_BKCUCX.Beckhoff_CXxxxx.Beckhoff_CXxxxxEK1122.A_0018_CX2040_EtherCAT_slave.Device_Status_Mapping.TxPdoToggle <-> Device Status Mapping/TxPdoToggle
//     PlcTask Inputs/GVL_iXlinker.EtherCAT_Master_BKCUCX.Beckhoff_CXxxxx.Beckhoff_CXxxxxEK1122.A_0018_CX2040_EtherCAT_slave.WcState.WcState <-> WcState/WcState
//     PlcTask Inputs/GVL_iXlinker.EtherCAT_Master_BKCUCX.Beckhoff_CXxxxx.Beckhoff_CXxxxxEK1122.A_0018_CX2040_EtherCAT_slave.WcState.InputToggle <-> WcState/InputToggle
//     PlcTask Inputs/GVL_iXlinker.EtherCAT_Master_BKCUCX.Beckhoff_CXxxxx.Beckhoff_CXxxxxEK1122.A_0018_CX2040_EtherCAT_slave.InfoData.AdsAddr <-> InfoData/AdsAddr
//     PlcTask Inputs/GVL_iXlinker.EtherCAT_Master_BKCUCX.Beckhoff_CXxxxx.Beckhoff_CXxxxxEK1122.A_0018_CX2040_EtherCAT_slave.InfoData.AoeNetId <-> InfoData/AoeNetId
//     PlcTask Inputs/GVL_iXlinker.EtherCAT_Master_BKCUCX.Beckhoff_CXxxxx.Beckhoff_CXxxxxEK1122.A_0018_CX2040_EtherCAT_slave.InfoData.State <-> InfoData/State
//   PLC/PLC Instance <-> EtherCAT Master BKCUCX/Beckhoff CXxxxx/Beckhoff CXxxxxEK1122/A_0019 (CX2040 EtherCAT slave)
//     PlcTask Inputs/GVL_iXlinker.EtherCAT_Master_BKCUCX.Beckhoff_CXxxxx.Beckhoff_CXxxxxEK1122.A_0019_CX2040_EtherCAT_slave.Device_Status_Mapping.TxPdoState <-> Device Status Mapping/TxPdoState
//     PlcTask Inputs/GVL_iXlinker.EtherCAT_Master_BKCUCX.Beckhoff_CXxxxx.Beckhoff_CXxxxxEK1122.A_0019_CX2040_EtherCAT_slave.Device_Status_Mapping.TxPdoToggle <-> Device Status Mapping/TxPdoToggle
//     PlcTask Inputs/GVL_iXlinker.EtherCAT_Master_BKCUCX.Beckhoff_CXxxxx.Beckhoff_CXxxxxEK1122.A_0019_CX2040_EtherCAT_slave.WcState.WcState <-> WcState/WcState
//     PlcTask Inputs/GVL_iXlinker.EtherCAT_Master_BKCUCX.Beckhoff_CXxxxx.Beckhoff_CXxxxxEK1122.A_0019_CX2040_EtherCAT_slave.WcState.InputToggle <-> WcState/InputToggle
//     PlcTask Inputs/GVL_iXlinker.EtherCAT_Master_BKCUCX.Beckhoff_CXxxxx.Beckhoff_CXxxxxEK1122.A_0019_CX2040_EtherCAT_slave.InfoData.AdsAddr <-> InfoData/AdsAddr
//     PlcTask Inputs/GVL_iXlinker.EtherCAT_Master_BKCUCX.Beckhoff_CXxxxx.Beckhoff_CXxxxxEK1122.A_0019_CX2040_EtherCAT_slave.InfoData.AoeNetId <-> InfoData/AoeNetId
//     PlcTask Inputs/GVL_iXlinker.EtherCAT_Master_BKCUCX.Beckhoff_CXxxxx.Beckhoff_CXxxxxEK1122.A_0019_CX2040_EtherCAT_slave.InfoData.State <-> InfoData/State
//   PLC/PLC Instance <-> EtherCAT Master BKCUCX/Beckhoff CXxxxx/Beckhoff CXxxxxEK1122/A_0020 (CX2040 EtherCAT slave)
//     PlcTask Inputs/GVL_iXlinker.EtherCAT_Master_BKCUCX.Beckhoff_CXxxxx.Beckhoff_CXxxxxEK1122.A_0020_CX2040_EtherCAT_slave.Device_Status_Mapping.TxPdoState <-> Device Status Mapping/TxPdoState
//     PlcTask Inputs/GVL_iXlinker.EtherCAT_Master_BKCUCX.Beckhoff_CXxxxx.Beckhoff_CXxxxxEK1122.A_0020_CX2040_EtherCAT_slave.Device_Status_Mapping.TxPdoToggle <-> Device Status Mapping/TxPdoToggle
//     PlcTask Inputs/GVL_iXlinker.EtherCAT_Master_BKCUCX.Beckhoff_CXxxxx.Beckhoff_CXxxxxEK1122.A_0020_CX2040_EtherCAT_slave.WcState.WcState <-> WcState/WcState
//     PlcTask Inputs/GVL_iXlinker.EtherCAT_Master_BKCUCX.Beckhoff_CXxxxx.Beckhoff_CXxxxxEK1122.A_0020_CX2040_EtherCAT_slave.WcState.InputToggle <-> WcState/InputToggle
//     PlcTask Inputs/GVL_iXlinker.EtherCAT_Master_BKCUCX.Beckhoff_CXxxxx.Beckhoff_CXxxxxEK1122.A_0020_CX2040_EtherCAT_slave.InfoData.AdsAddr <-> InfoData/AdsAddr
//     PlcTask Inputs/GVL_iXlinker.EtherCAT_Master_BKCUCX.Beckhoff_CXxxxx.Beckhoff_CXxxxxEK1122.A_0020_CX2040_EtherCAT_slave.InfoData.AoeNetId <-> InfoData/AoeNetId
//     PlcTask Inputs/GVL_iXlinker.EtherCAT_Master_BKCUCX.Beckhoff_CXxxxx.Beckhoff_CXxxxxEK1122.A_0020_CX2040_EtherCAT_slave.InfoData.State <-> InfoData/State
//   PLC/PLC Instance <-> EtherCAT Master BKCUCX/Beckhoff CXxxxx/Beckhoff CXxxxxEK1122/A_0021 (CX2042 EtherCAT slave)
//     PlcTask Inputs/GVL_iXlinker.EtherCAT_Master_BKCUCX.Beckhoff_CXxxxx.Beckhoff_CXxxxxEK1122.A_0021_CX2042_EtherCAT_slave.Device_Status_Mapping.TxPdoState <-> Device Status Mapping/TxPdoState
//     PlcTask Inputs/GVL_iXlinker.EtherCAT_Master_BKCUCX.Beckhoff_CXxxxx.Beckhoff_CXxxxxEK1122.A_0021_CX2042_EtherCAT_slave.Device_Status_Mapping.TxPdoToggle <-> Device Status Mapping/TxPdoToggle
//     PlcTask Inputs/GVL_iXlinker.EtherCAT_Master_BKCUCX.Beckhoff_CXxxxx.Beckhoff_CXxxxxEK1122.A_0021_CX2042_EtherCAT_slave.WcState.WcState <-> WcState/WcState
//     PlcTask Inputs/GVL_iXlinker.EtherCAT_Master_BKCUCX.Beckhoff_CXxxxx.Beckhoff_CXxxxxEK1122.A_0021_CX2042_EtherCAT_slave.WcState.InputToggle <-> WcState/InputToggle
//     PlcTask Inputs/GVL_iXlinker.EtherCAT_Master_BKCUCX.Beckhoff_CXxxxx.Beckhoff_CXxxxxEK1122.A_0021_CX2042_EtherCAT_slave.InfoData.AdsAddr <-> InfoData/AdsAddr
//     PlcTask Inputs/GVL_iXlinker.EtherCAT_Master_BKCUCX.Beckhoff_CXxxxx.Beckhoff_CXxxxxEK1122.A_0021_CX2042_EtherCAT_slave.InfoData.AoeNetId <-> InfoData/AoeNetId
//     PlcTask Inputs/GVL_iXlinker.EtherCAT_Master_BKCUCX.Beckhoff_CXxxxx.Beckhoff_CXxxxxEK1122.A_0021_CX2042_EtherCAT_slave.InfoData.State <-> InfoData/State
//   PLC/PLC Instance <-> EtherCAT Master BKCUCX/Beckhoff CXxxxx/Beckhoff CXxxxxEK1122/A_0022 (CX2043 EtherCAT slave)
//     PlcTask Inputs/GVL_iXlinker.EtherCAT_Master_BKCUCX.Beckhoff_CXxxxx.Beckhoff_CXxxxxEK1122.A_0022_CX2043_EtherCAT_slave.Device_Status_Mapping.TxPdoState <-> Device Status Mapping/TxPdoState
//     PlcTask Inputs/GVL_iXlinker.EtherCAT_Master_BKCUCX.Beckhoff_CXxxxx.Beckhoff_CXxxxxEK1122.A_0022_CX2043_EtherCAT_slave.Device_Status_Mapping.TxPdoToggle <-> Device Status Mapping/TxPdoToggle
//     PlcTask Inputs/GVL_iXlinker.EtherCAT_Master_BKCUCX.Beckhoff_CXxxxx.Beckhoff_CXxxxxEK1122.A_0022_CX2043_EtherCAT_slave.WcState.WcState <-> WcState/WcState
//     PlcTask Inputs/GVL_iXlinker.EtherCAT_Master_BKCUCX.Beckhoff_CXxxxx.Beckhoff_CXxxxxEK1122.A_0022_CX2043_EtherCAT_slave.WcState.InputToggle <-> WcState/InputToggle
//     PlcTask Inputs/GVL_iXlinker.EtherCAT_Master_BKCUCX.Beckhoff_CXxxxx.Beckhoff_CXxxxxEK1122.A_0022_CX2043_EtherCAT_slave.InfoData.AdsAddr <-> InfoData/AdsAddr
//     PlcTask Inputs/GVL_iXlinker.EtherCAT_Master_BKCUCX.Beckhoff_CXxxxx.Beckhoff_CXxxxxEK1122.A_0022_CX2043_EtherCAT_slave.InfoData.AoeNetId <-> InfoData/AoeNetId
//     PlcTask Inputs/GVL_iXlinker.EtherCAT_Master_BKCUCX.Beckhoff_CXxxxx.Beckhoff_CXxxxxEK1122.A_0022_CX2043_EtherCAT_slave.InfoData.State <-> InfoData/State
//   PLC/PLC Instance <-> EtherCAT Master BKCUCX/Beckhoff CXxxxx/Beckhoff CXxxxxEK1122/A_0023 (CX2062 EtherCAT slave)
//     PlcTask Inputs/GVL_iXlinker.EtherCAT_Master_BKCUCX.Beckhoff_CXxxxx.Beckhoff_CXxxxxEK1122.A_0023_CX2062_EtherCAT_slave.Device_Status_Mapping.TxPdoState <-> Device Status Mapping/TxPdoState
//     PlcTask Inputs/GVL_iXlinker.EtherCAT_Master_BKCUCX.Beckhoff_CXxxxx.Beckhoff_CXxxxxEK1122.A_0023_CX2062_EtherCAT_slave.Device_Status_Mapping.TxPdoToggle <-> Device Status Mapping/TxPdoToggle
//     PlcTask Inputs/GVL_iXlinker.EtherCAT_Master_BKCUCX.Beckhoff_CXxxxx.Beckhoff_CXxxxxEK1122.A_0023_CX2062_EtherCAT_slave.WcState.WcState <-> WcState/WcState
//     PlcTask Inputs/GVL_iXlinker.EtherCAT_Master_BKCUCX.Beckhoff_CXxxxx.Beckhoff_CXxxxxEK1122.A_0023_CX2062_EtherCAT_slave.WcState.InputToggle <-> WcState/InputToggle
//     PlcTask Inputs/GVL_iXlinker.EtherCAT_Master_BKCUCX.Beckhoff_CXxxxx.Beckhoff_CXxxxxEK1122.A_0023_CX2062_EtherCAT_slave.InfoData.AdsAddr <-> InfoData/AdsAddr
//     PlcTask Inputs/GVL_iXlinker.EtherCAT_Master_BKCUCX.Beckhoff_CXxxxx.Beckhoff_CXxxxxEK1122.A_0023_CX2062_EtherCAT_slave.InfoData.AoeNetId <-> InfoData/AoeNetId
//     PlcTask Inputs/GVL_iXlinker.EtherCAT_Master_BKCUCX.Beckhoff_CXxxxx.Beckhoff_CXxxxxEK1122.A_0023_CX2062_EtherCAT_slave.InfoData.State <-> InfoData/State
//   PLC/PLC Instance <-> EtherCAT Master BKCUCX/Beckhoff CXxxxx/Beckhoff CXxxxxEK1122/A_0024 (CX2072 EtherCAT slave)
//     PlcTask Inputs/GVL_iXlinker.EtherCAT_Master_BKCUCX.Beckhoff_CXxxxx.Beckhoff_CXxxxxEK1122.A_0024_CX2072_EtherCAT_slave.Device_Status_Mapping.TxPdoState <-> Device Status Mapping/TxPdoState
//     PlcTask Inputs/GVL_iXlinker.EtherCAT_Master_BKCUCX.Beckhoff_CXxxxx.Beckhoff_CXxxxxEK1122.A_0024_CX2072_EtherCAT_slave.Device_Status_Mapping.TxPdoToggle <-> Device Status Mapping/TxPdoToggle
//     PlcTask Inputs/GVL_iXlinker.EtherCAT_Master_BKCUCX.Beckhoff_CXxxxx.Beckhoff_CXxxxxEK1122.A_0024_CX2072_EtherCAT_slave.WcState.WcState <-> WcState/WcState
//     PlcTask Inputs/GVL_iXlinker.EtherCAT_Master_BKCUCX.Beckhoff_CXxxxx.Beckhoff_CXxxxxEK1122.A_0024_CX2072_EtherCAT_slave.WcState.InputToggle <-> WcState/InputToggle
//     PlcTask Inputs/GVL_iXlinker.EtherCAT_Master_BKCUCX.Beckhoff_CXxxxx.Beckhoff_CXxxxxEK1122.A_0024_CX2072_EtherCAT_slave.InfoData.AdsAddr <-> InfoData/AdsAddr
//     PlcTask Inputs/GVL_iXlinker.EtherCAT_Master_BKCUCX.Beckhoff_CXxxxx.Beckhoff_CXxxxxEK1122.A_0024_CX2072_EtherCAT_slave.InfoData.AoeNetId <-> InfoData/AoeNetId
//     PlcTask Inputs/GVL_iXlinker.EtherCAT_Master_BKCUCX.Beckhoff_CXxxxx.Beckhoff_CXxxxxEK1122.A_0024_CX2072_EtherCAT_slave.InfoData.State <-> InfoData/State
//   PLC/PLC Instance <-> EtherCAT Master BKCUCX/Beckhoff CXxxxx/Beckhoff CXxxxxEK1122/A_0025 (CX9020 EtherCAT slave)
//     PlcTask Inputs/GVL_iXlinker.EtherCAT_Master_BKCUCX.Beckhoff_CXxxxx.Beckhoff_CXxxxxEK1122.A_0025_CX9020_EtherCAT_slave.Device_Status_Mapping.TxPdoState <-> Device Status Mapping/TxPdoState
//     PlcTask Inputs/GVL_iXlinker.EtherCAT_Master_BKCUCX.Beckhoff_CXxxxx.Beckhoff_CXxxxxEK1122.A_0025_CX9020_EtherCAT_slave.Device_Status_Mapping.TxPdoToggle <-> Device Status Mapping/TxPdoToggle
//     PlcTask Inputs/GVL_iXlinker.EtherCAT_Master_BKCUCX.Beckhoff_CXxxxx.Beckhoff_CXxxxxEK1122.A_0025_CX9020_EtherCAT_slave.WcState.WcState <-> WcState/WcState
//     PlcTask Inputs/GVL_iXlinker.EtherCAT_Master_BKCUCX.Beckhoff_CXxxxx.Beckhoff_CXxxxxEK1122.A_0025_CX9020_EtherCAT_slave.WcState.InputToggle <-> WcState/InputToggle
//     PlcTask Inputs/GVL_iXlinker.EtherCAT_Master_BKCUCX.Beckhoff_CXxxxx.Beckhoff_CXxxxxEK1122.A_0025_CX9020_EtherCAT_slave.InfoData.AdsAddr <-> InfoData/AdsAddr
//     PlcTask Inputs/GVL_iXlinker.EtherCAT_Master_BKCUCX.Beckhoff_CXxxxx.Beckhoff_CXxxxxEK1122.A_0025_CX9020_EtherCAT_slave.InfoData.AoeNetId <-> InfoData/AoeNetId
//     PlcTask Inputs/GVL_iXlinker.EtherCAT_Master_BKCUCX.Beckhoff_CXxxxx.Beckhoff_CXxxxxEK1122.A_0025_CX9020_EtherCAT_slave.InfoData.State <-> InfoData/State
//   PLC/PLC Instance <-> EtherCAT Master BKCUCX/Beckhoff CXxxxx/Beckhoff CXxxxxEK1122/A_0026 (CX9020 EtherCAT slave)
//     PlcTask Inputs/GVL_iXlinker.EtherCAT_Master_BKCUCX.Beckhoff_CXxxxx.Beckhoff_CXxxxxEK1122.A_0026_CX9020_EtherCAT_slave.Device_Status_Mapping.TxPdoState <-> Device Status Mapping/TxPdoState
//     PlcTask Inputs/GVL_iXlinker.EtherCAT_Master_BKCUCX.Beckhoff_CXxxxx.Beckhoff_CXxxxxEK1122.A_0026_CX9020_EtherCAT_slave.Device_Status_Mapping.TxPdoToggle <-> Device Status Mapping/TxPdoToggle
//     PlcTask Inputs/GVL_iXlinker.EtherCAT_Master_BKCUCX.Beckhoff_CXxxxx.Beckhoff_CXxxxxEK1122.A_0026_CX9020_EtherCAT_slave.WcState.WcState <-> WcState/WcState
//     PlcTask Inputs/GVL_iXlinker.EtherCAT_Master_BKCUCX.Beckhoff_CXxxxx.Beckhoff_CXxxxxEK1122.A_0026_CX9020_EtherCAT_slave.WcState.InputToggle <-> WcState/InputToggle
//     PlcTask Inputs/GVL_iXlinker.EtherCAT_Master_BKCUCX.Beckhoff_CXxxxx.Beckhoff_CXxxxxEK1122.A_0026_CX9020_EtherCAT_slave.InfoData.AdsAddr <-> InfoData/AdsAddr
//     PlcTask Inputs/GVL_iXlinker.EtherCAT_Master_BKCUCX.Beckhoff_CXxxxx.Beckhoff_CXxxxxEK1122.A_0026_CX9020_EtherCAT_slave.InfoData.AoeNetId <-> InfoData/AoeNetId
//     PlcTask Inputs/GVL_iXlinker.EtherCAT_Master_BKCUCX.Beckhoff_CXxxxx.Beckhoff_CXxxxxEK1122.A_0026_CX9020_EtherCAT_slave.InfoData.State <-> InfoData/State
//   PLC/PLC Instance <-> EtherCAT Master BKCUCX/Beckhoff CXxxxx/Beckhoff CXxxxxEK1122/A_0027 (CX5120 EtherCAT slave)
//     PlcTask Inputs/GVL_iXlinker.EtherCAT_Master_BKCUCX.Beckhoff_CXxxxx.Beckhoff_CXxxxxEK1122.A_0027_CX5120_EtherCAT_slave.Device_Status_Mapping.TxPdoState <-> Device Status Mapping/TxPdoState
//     PlcTask Inputs/GVL_iXlinker.EtherCAT_Master_BKCUCX.Beckhoff_CXxxxx.Beckhoff_CXxxxxEK1122.A_0027_CX5120_EtherCAT_slave.Device_Status_Mapping.TxPdoToggle <-> Device Status Mapping/TxPdoToggle
//     PlcTask Inputs/GVL_iXlinker.EtherCAT_Master_BKCUCX.Beckhoff_CXxxxx.Beckhoff_CXxxxxEK1122.A_0027_CX5120_EtherCAT_slave.WcState.WcState <-> WcState/WcState
//     PlcTask Inputs/GVL_iXlinker.EtherCAT_Master_BKCUCX.Beckhoff_CXxxxx.Beckhoff_CXxxxxEK1122.A_0027_CX5120_EtherCAT_slave.WcState.InputToggle <-> WcState/InputToggle
//     PlcTask Inputs/GVL_iXlinker.EtherCAT_Master_BKCUCX.Beckhoff_CXxxxx.Beckhoff_CXxxxxEK1122.A_0027_CX5120_EtherCAT_slave.InfoData.AdsAddr <-> InfoData/AdsAddr
//     PlcTask Inputs/GVL_iXlinker.EtherCAT_Master_BKCUCX.Beckhoff_CXxxxx.Beckhoff_CXxxxxEK1122.A_0027_CX5120_EtherCAT_slave.InfoData.AoeNetId <-> InfoData/AoeNetId
//     PlcTask Inputs/GVL_iXlinker.EtherCAT_Master_BKCUCX.Beckhoff_CXxxxx.Beckhoff_CXxxxxEK1122.A_0027_CX5120_EtherCAT_slave.InfoData.State <-> InfoData/State
//   PLC/PLC Instance <-> EtherCAT Master BKCUCX/Beckhoff CXxxxx/Beckhoff CXxxxxEK1122/A_0028 (CX5130 EtherCAT slave)
//     PlcTask Inputs/GVL_iXlinker.EtherCAT_Master_BKCUCX.Beckhoff_CXxxxx.Beckhoff_CXxxxxEK1122.A_0028_CX5130_EtherCAT_slave.Device_Status_Mapping.TxPdoState <-> Device Status Mapping/TxPdoState
//     PlcTask Inputs/GVL_iXlinker.EtherCAT_Master_BKCUCX.Beckhoff_CXxxxx.Beckhoff_CXxxxxEK1122.A_0028_CX5130_EtherCAT_slave.Device_Status_Mapping.TxPdoToggle <-> Device Status Mapping/TxPdoToggle
//     PlcTask Inputs/GVL_iXlinker.EtherCAT_Master_BKCUCX.Beckhoff_CXxxxx.Beckhoff_CXxxxxEK1122.A_0028_CX5130_EtherCAT_slave.WcState.WcState <-> WcState/WcState
//     PlcTask Inputs/GVL_iXlinker.EtherCAT_Master_BKCUCX.Beckhoff_CXxxxx.Beckhoff_CXxxxxEK1122.A_0028_CX5130_EtherCAT_slave.WcState.InputToggle <-> WcState/InputToggle
//     PlcTask Inputs/GVL_iXlinker.EtherCAT_Master_BKCUCX.Beckhoff_CXxxxx.Beckhoff_CXxxxxEK1122.A_0028_CX5130_EtherCAT_slave.InfoData.AdsAddr <-> InfoData/AdsAddr
//     PlcTask Inputs/GVL_iXlinker.EtherCAT_Master_BKCUCX.Beckhoff_CXxxxx.Beckhoff_CXxxxxEK1122.A_0028_CX5130_EtherCAT_slave.InfoData.AoeNetId <-> InfoData/AoeNetId
//     PlcTask Inputs/GVL_iXlinker.EtherCAT_Master_BKCUCX.Beckhoff_CXxxxx.Beckhoff_CXxxxxEK1122.A_0028_CX5130_EtherCAT_slave.InfoData.State <-> InfoData/State
//   PLC/PLC Instance <-> EtherCAT Master BKCUCX/Beckhoff CXxxxx/Beckhoff CXxxxxEK1122/A_0029 (CX5140 EtherCAT slave)
//     PlcTask Inputs/GVL_iXlinker.EtherCAT_Master_BKCUCX.Beckhoff_CXxxxx.Beckhoff_CXxxxxEK1122.A_0029_CX5140_EtherCAT_slave.Device_Status_Mapping.TxPdoState <-> Device Status Mapping/TxPdoState
//     PlcTask Inputs/GVL_iXlinker.EtherCAT_Master_BKCUCX.Beckhoff_CXxxxx.Beckhoff_CXxxxxEK1122.A_0029_CX5140_EtherCAT_slave.Device_Status_Mapping.TxPdoToggle <-> Device Status Mapping/TxPdoToggle
//     PlcTask Inputs/GVL_iXlinker.EtherCAT_Master_BKCUCX.Beckhoff_CXxxxx.Beckhoff_CXxxxxEK1122.A_0029_CX5140_EtherCAT_slave.WcState.WcState <-> WcState/WcState
//     PlcTask Inputs/GVL_iXlinker.EtherCAT_Master_BKCUCX.Beckhoff_CXxxxx.Beckhoff_CXxxxxEK1122.A_0029_CX5140_EtherCAT_slave.WcState.InputToggle <-> WcState/InputToggle
//     PlcTask Inputs/GVL_iXlinker.EtherCAT_Master_BKCUCX.Beckhoff_CXxxxx.Beckhoff_CXxxxxEK1122.A_0029_CX5140_EtherCAT_slave.InfoData.AdsAddr <-> InfoData/AdsAddr
//     PlcTask Inputs/GVL_iXlinker.EtherCAT_Master_BKCUCX.Beckhoff_CXxxxx.Beckhoff_CXxxxxEK1122.A_0029_CX5140_EtherCAT_slave.InfoData.AoeNetId <-> InfoData/AoeNetId
//     PlcTask Inputs/GVL_iXlinker.EtherCAT_Master_BKCUCX.Beckhoff_CXxxxx.Beckhoff_CXxxxxEK1122.A_0029_CX5140_EtherCAT_slave.InfoData.State <-> InfoData/State
//   PLC/PLC Instance <-> EtherCAT Master BKCUCX/Beckhoff CXxxxx/Beckhoff CXxxxxEK1122/A_0030 (CX5230 EtherCAT slave)
//     PlcTask Inputs/GVL_iXlinker.EtherCAT_Master_BKCUCX.Beckhoff_CXxxxx.Beckhoff_CXxxxxEK1122.A_0030_CX5230_EtherCAT_slave.Device_Status_Mapping.TxPdoState <-> Device Status Mapping/TxPdoState
//     PlcTask Inputs/GVL_iXlinker.EtherCAT_Master_BKCUCX.Beckhoff_CXxxxx.Beckhoff_CXxxxxEK1122.A_0030_CX5230_EtherCAT_slave.Device_Status_Mapping.TxPdoToggle <-> Device Status Mapping/TxPdoToggle
//     PlcTask Inputs/GVL_iXlinker.EtherCAT_Master_BKCUCX.Beckhoff_CXxxxx.Beckhoff_CXxxxxEK1122.A_0030_CX5230_EtherCAT_slave.WcState.WcState <-> WcState/WcState
//     PlcTask Inputs/GVL_iXlinker.EtherCAT_Master_BKCUCX.Beckhoff_CXxxxx.Beckhoff_CXxxxxEK1122.A_0030_CX5230_EtherCAT_slave.WcState.InputToggle <-> WcState/InputToggle
//     PlcTask Inputs/GVL_iXlinker.EtherCAT_Master_BKCUCX.Beckhoff_CXxxxx.Beckhoff_CXxxxxEK1122.A_0030_CX5230_EtherCAT_slave.InfoData.AdsAddr <-> InfoData/AdsAddr
//     PlcTask Inputs/GVL_iXlinker.EtherCAT_Master_BKCUCX.Beckhoff_CXxxxx.Beckhoff_CXxxxxEK1122.A_0030_CX5230_EtherCAT_slave.InfoData.AoeNetId <-> InfoData/AoeNetId
//     PlcTask Inputs/GVL_iXlinker.EtherCAT_Master_BKCUCX.Beckhoff_CXxxxx.Beckhoff_CXxxxxEK1122.A_0030_CX5230_EtherCAT_slave.InfoData.State <-> InfoData/State
//   PLC/PLC Instance <-> EtherCAT Master BKCUCX/Beckhoff CXxxxx/Beckhoff CXxxxxEK1122/A_0031 (CX5240 EtherCAT slave)
//     PlcTask Inputs/GVL_iXlinker.EtherCAT_Master_BKCUCX.Beckhoff_CXxxxx.Beckhoff_CXxxxxEK1122.A_0031_CX5240_EtherCAT_slave.Device_Status_Mapping.TxPdoState <-> Device Status Mapping/TxPdoState
//     PlcTask Inputs/GVL_iXlinker.EtherCAT_Master_BKCUCX.Beckhoff_CXxxxx.Beckhoff_CXxxxxEK1122.A_0031_CX5240_EtherCAT_slave.Device_Status_Mapping.TxPdoToggle <-> Device Status Mapping/TxPdoToggle
//     PlcTask Inputs/GVL_iXlinker.EtherCAT_Master_BKCUCX.Beckhoff_CXxxxx.Beckhoff_CXxxxxEK1122.A_0031_CX5240_EtherCAT_slave.WcState.WcState <-> WcState/WcState
//     PlcTask Inputs/GVL_iXlinker.EtherCAT_Master_BKCUCX.Beckhoff_CXxxxx.Beckhoff_CXxxxxEK1122.A_0031_CX5240_EtherCAT_slave.WcState.InputToggle <-> WcState/InputToggle
//     PlcTask Inputs/GVL_iXlinker.EtherCAT_Master_BKCUCX.Beckhoff_CXxxxx.Beckhoff_CXxxxxEK1122.A_0031_CX5240_EtherCAT_slave.InfoData.AdsAddr <-> InfoData/AdsAddr
//     PlcTask Inputs/GVL_iXlinker.EtherCAT_Master_BKCUCX.Beckhoff_CXxxxx.Beckhoff_CXxxxxEK1122.A_0031_CX5240_EtherCAT_slave.InfoData.AoeNetId <-> InfoData/AoeNetId
//     PlcTask Inputs/GVL_iXlinker.EtherCAT_Master_BKCUCX.Beckhoff_CXxxxx.Beckhoff_CXxxxxEK1122.A_0031_CX5240_EtherCAT_slave.InfoData.State <-> InfoData/State
//   PLC/PLC Instance <-> EtherCAT Master BKCUCX/Beckhoff CXxxxx/Beckhoff CXxxxxEK1122/A_0002(CX1100-0004-0001)
//     PlcTask Inputs/GVL_iXlinker.EtherCAT_Master_BKCUCX.Beckhoff_CXxxxx.Beckhoff_CXxxxxEK1122.A_0002_CX1100_0004_0001.InfoData.State <-> InfoData/State
//   PLC/PLC Instance <-> EtherCAT Master BKCUCX/TcTerminals210_EK1100_1
//     PlcTask Inputs/GVL_iXlinker.EtherCAT_Master_BKCUCX.TcTerminals210_EK1100_1.InfoData.State <-> InfoData/State
//   PLC/PLC Instance <-> EtherCAT Master BKCUCX/TcTerminals210_EK1100_1/TcTerminals210_1BK1250
//     PlcTask Inputs/GVL_iXlinker.EtherCAT_Master_BKCUCX.TcTerminals210_EK1100_1.TcTerminals210_1BK1250.Inputs.CouplerState <-> Inputs/CouplerState
//     PlcTask Inputs/GVL_iXlinker.EtherCAT_Master_BKCUCX.TcTerminals210_EK1100_1.TcTerminals210_1BK1250.Outputs.CouplerCtrl <-> Outputs/CouplerCtrl
//     PlcTask Inputs/GVL_iXlinker.EtherCAT_Master_BKCUCX.TcTerminals210_EK1100_1.TcTerminals210_1BK1250.WcState.WcState <-> WcState/WcState
//     PlcTask Inputs/GVL_iXlinker.EtherCAT_Master_BKCUCX.TcTerminals210_EK1100_1.TcTerminals210_1BK1250.WcState.InputToggle <-> WcState/InputToggle
//     PlcTask Inputs/GVL_iXlinker.EtherCAT_Master_BKCUCX.TcTerminals210_EK1100_1.TcTerminals210_1BK1250.InfoData.AdsAddr <-> InfoData/AdsAddr
//     PlcTask Inputs/GVL_iXlinker.EtherCAT_Master_BKCUCX.TcTerminals210_EK1100_1.TcTerminals210_1BK1250.InfoData.AoeNetId <-> InfoData/AoeNetId
//     PlcTask Inputs/GVL_iXlinker.EtherCAT_Master_BKCUCX.TcTerminals210_EK1100_1.TcTerminals210_1BK1250.InfoData.State <-> InfoData/State
//   PLC/PLC Instance <-> EtherCAT Master BKCUCX/TcTerminals210_EK1100_1/TcTerminals210_1BK1250/A_0006(CP9940-0001 40 Ch. Input)
//     PlcTask Inputs/GVL_iXlinker.EtherCAT_Master_BKCUCX.TcTerminals210_EK1100_1.TcTerminals210_1BK1250.A_0006_CP9940_0001_40_Ch_Input.Channel_1.Key_1 <-> Channel 1/Key 1
//     PlcTask Inputs/GVL_iXlinker.EtherCAT_Master_BKCUCX.TcTerminals210_EK1100_1.TcTerminals210_1BK1250.A_0006_CP9940_0001_40_Ch_Input.Channel_1.Key_2 <-> Channel 1/Key 2
//     PlcTask Inputs/GVL_iXlinker.EtherCAT_Master_BKCUCX.TcTerminals210_EK1100_1.TcTerminals210_1BK1250.A_0006_CP9940_0001_40_Ch_Input.Channel_1.Key_3 <-> Channel 1/Key 3
//     PlcTask Inputs/GVL_iXlinker.EtherCAT_Master_BKCUCX.TcTerminals210_EK1100_1.TcTerminals210_1BK1250.A_0006_CP9940_0001_40_Ch_Input.Channel_1.Key_4 <-> Channel 1/Key 4
//     PlcTask Inputs/GVL_iXlinker.EtherCAT_Master_BKCUCX.TcTerminals210_EK1100_1.TcTerminals210_1BK1250.A_0006_CP9940_0001_40_Ch_Input.Channel_1.Key_5 <-> Channel 1/Key 5
//     PlcTask Inputs/GVL_iXlinker.EtherCAT_Master_BKCUCX.TcTerminals210_EK1100_1.TcTerminals210_1BK1250.A_0006_CP9940_0001_40_Ch_Input.Channel_1.Key_6 <-> Channel 1/Key 6
//     PlcTask Inputs/GVL_iXlinker.EtherCAT_Master_BKCUCX.TcTerminals210_EK1100_1.TcTerminals210_1BK1250.A_0006_CP9940_0001_40_Ch_Input.Channel_1.Key_7 <-> Channel 1/Key 7
//     PlcTask Inputs/GVL_iXlinker.EtherCAT_Master_BKCUCX.TcTerminals210_EK1100_1.TcTerminals210_1BK1250.A_0006_CP9940_0001_40_Ch_Input.Channel_1.Key_8 <-> Channel 1/Key 8
//     PlcTask Inputs/GVL_iXlinker.EtherCAT_Master_BKCUCX.TcTerminals210_EK1100_1.TcTerminals210_1BK1250.A_0006_CP9940_0001_40_Ch_Input.Channel_1.Key_9 <-> Channel 1/Key 9
//     PlcTask Inputs/GVL_iXlinker.EtherCAT_Master_BKCUCX.TcTerminals210_EK1100_1.TcTerminals210_1BK1250.A_0006_CP9940_0001_40_Ch_Input.Channel_1.Key_10 <-> Channel 1/Key 10
//     PlcTask Inputs/GVL_iXlinker.EtherCAT_Master_BKCUCX.TcTerminals210_EK1100_1.TcTerminals210_1BK1250.A_0006_CP9940_0001_40_Ch_Input.Channel_1.Key_11 <-> Channel 1/Key 11
//     PlcTask Inputs/GVL_iXlinker.EtherCAT_Master_BKCUCX.TcTerminals210_EK1100_1.TcTerminals210_1BK1250.A_0006_CP9940_0001_40_Ch_Input.Channel_1.Key_12 <-> Channel 1/Key 12
//     PlcTask Inputs/GVL_iXlinker.EtherCAT_Master_BKCUCX.TcTerminals210_EK1100_1.TcTerminals210_1BK1250.A_0006_CP9940_0001_40_Ch_Input.Channel_1.Key_13 <-> Channel 1/Key 13
//     PlcTask Inputs/GVL_iXlinker.EtherCAT_Master_BKCUCX.TcTerminals210_EK1100_1.TcTerminals210_1BK1250.A_0006_CP9940_0001_40_Ch_Input.Channel_1.Key_14 <-> Channel 1/Key 14
//     PlcTask Inputs/GVL_iXlinker.EtherCAT_Master_BKCUCX.TcTerminals210_EK1100_1.TcTerminals210_1BK1250.A_0006_CP9940_0001_40_Ch_Input.Channel_1.Key_15 <-> Channel 1/Key 15
//     PlcTask Inputs/GVL_iXlinker.EtherCAT_Master_BKCUCX.TcTerminals210_EK1100_1.TcTerminals210_1BK1250.A_0006_CP9940_0001_40_Ch_Input.Channel_1.Key_16 <-> Channel 1/Key 16
//     PlcTask Inputs/GVL_iXlinker.EtherCAT_Master_BKCUCX.TcTerminals210_EK1100_1.TcTerminals210_1BK1250.A_0006_CP9940_0001_40_Ch_Input.Channel_1.Key_17 <-> Channel 1/Key 17
//     PlcTask Inputs/GVL_iXlinker.EtherCAT_Master_BKCUCX.TcTerminals210_EK1100_1.TcTerminals210_1BK1250.A_0006_CP9940_0001_40_Ch_Input.Channel_1.Key_18 <-> Channel 1/Key 18
//     PlcTask Inputs/GVL_iXlinker.EtherCAT_Master_BKCUCX.TcTerminals210_EK1100_1.TcTerminals210_1BK1250.A_0006_CP9940_0001_40_Ch_Input.Channel_1.Key_19 <-> Channel 1/Key 19
//     PlcTask Inputs/GVL_iXlinker.EtherCAT_Master_BKCUCX.TcTerminals210_EK1100_1.TcTerminals210_1BK1250.A_0006_CP9940_0001_40_Ch_Input.Channel_1.Key_20 <-> Channel 1/Key 20
//     PlcTask Inputs/GVL_iXlinker.EtherCAT_Master_BKCUCX.TcTerminals210_EK1100_1.TcTerminals210_1BK1250.A_0006_CP9940_0001_40_Ch_Input.Channel_1.Key_21 <-> Channel 1/Key 21
//     PlcTask Inputs/GVL_iXlinker.EtherCAT_Master_BKCUCX.TcTerminals210_EK1100_1.TcTerminals210_1BK1250.A_0006_CP9940_0001_40_Ch_Input.Channel_1.Key_22 <-> Channel 1/Key 22
//     PlcTask Inputs/GVL_iXlinker.EtherCAT_Master_BKCUCX.TcTerminals210_EK1100_1.TcTerminals210_1BK1250.A_0006_CP9940_0001_40_Ch_Input.Channel_1.Key_23 <-> Channel 1/Key 23
//     PlcTask Inputs/GVL_iXlinker.EtherCAT_Master_BKCUCX.TcTerminals210_EK1100_1.TcTerminals210_1BK1250.A_0006_CP9940_0001_40_Ch_Input.Channel_1.Key_24 <-> Channel 1/Key 24
//     PlcTask Inputs/GVL_iXlinker.EtherCAT_Master_BKCUCX.TcTerminals210_EK1100_1.TcTerminals210_1BK1250.A_0006_CP9940_0001_40_Ch_Input.Channel_1.Key_25 <-> Channel 1/Key 25
//     PlcTask Inputs/GVL_iXlinker.EtherCAT_Master_BKCUCX.TcTerminals210_EK1100_1.TcTerminals210_1BK1250.A_0006_CP9940_0001_40_Ch_Input.Channel_1.Key_26 <-> Channel 1/Key 26
//     PlcTask Inputs/GVL_iXlinker.EtherCAT_Master_BKCUCX.TcTerminals210_EK1100_1.TcTerminals210_1BK1250.A_0006_CP9940_0001_40_Ch_Input.Channel_1.Key_27 <-> Channel 1/Key 27
//     PlcTask Inputs/GVL_iXlinker.EtherCAT_Master_BKCUCX.TcTerminals210_EK1100_1.TcTerminals210_1BK1250.A_0006_CP9940_0001_40_Ch_Input.Channel_1.Key_28 <-> Channel 1/Key 28
//     PlcTask Inputs/GVL_iXlinker.EtherCAT_Master_BKCUCX.TcTerminals210_EK1100_1.TcTerminals210_1BK1250.A_0006_CP9940_0001_40_Ch_Input.Channel_1.Key_29 <-> Channel 1/Key 29
//     PlcTask Inputs/GVL_iXlinker.EtherCAT_Master_BKCUCX.TcTerminals210_EK1100_1.TcTerminals210_1BK1250.A_0006_CP9940_0001_40_Ch_Input.Channel_1.Key_30 <-> Channel 1/Key 30
//     PlcTask Inputs/GVL_iXlinker.EtherCAT_Master_BKCUCX.TcTerminals210_EK1100_1.TcTerminals210_1BK1250.A_0006_CP9940_0001_40_Ch_Input.Channel_1.Key_31 <-> Channel 1/Key 31
//     PlcTask Inputs/GVL_iXlinker.EtherCAT_Master_BKCUCX.TcTerminals210_EK1100_1.TcTerminals210_1BK1250.A_0006_CP9940_0001_40_Ch_Input.Channel_1.Key_32 <-> Channel 1/Key 32
//     PlcTask Inputs/GVL_iXlinker.EtherCAT_Master_BKCUCX.TcTerminals210_EK1100_1.TcTerminals210_1BK1250.A_0006_CP9940_0001_40_Ch_Input.Channel_1.Key_33 <-> Channel 1/Key 33
//     PlcTask Inputs/GVL_iXlinker.EtherCAT_Master_BKCUCX.TcTerminals210_EK1100_1.TcTerminals210_1BK1250.A_0006_CP9940_0001_40_Ch_Input.Channel_1.Key_34 <-> Channel 1/Key 34
//     PlcTask Inputs/GVL_iXlinker.EtherCAT_Master_BKCUCX.TcTerminals210_EK1100_1.TcTerminals210_1BK1250.A_0006_CP9940_0001_40_Ch_Input.Channel_1.Key_35 <-> Channel 1/Key 35
//     PlcTask Inputs/GVL_iXlinker.EtherCAT_Master_BKCUCX.TcTerminals210_EK1100_1.TcTerminals210_1BK1250.A_0006_CP9940_0001_40_Ch_Input.Channel_1.Key_36 <-> Channel 1/Key 36
//     PlcTask Inputs/GVL_iXlinker.EtherCAT_Master_BKCUCX.TcTerminals210_EK1100_1.TcTerminals210_1BK1250.A_0006_CP9940_0001_40_Ch_Input.Channel_1.Key_37 <-> Channel 1/Key 37
//     PlcTask Inputs/GVL_iXlinker.EtherCAT_Master_BKCUCX.TcTerminals210_EK1100_1.TcTerminals210_1BK1250.A_0006_CP9940_0001_40_Ch_Input.Channel_1.Key_38 <-> Channel 1/Key 38
//     PlcTask Inputs/GVL_iXlinker.EtherCAT_Master_BKCUCX.TcTerminals210_EK1100_1.TcTerminals210_1BK1250.A_0006_CP9940_0001_40_Ch_Input.Channel_1.Key_39 <-> Channel 1/Key 39
//     PlcTask Inputs/GVL_iXlinker.EtherCAT_Master_BKCUCX.TcTerminals210_EK1100_1.TcTerminals210_1BK1250.A_0006_CP9940_0001_40_Ch_Input.Channel_1.Key_40 <-> Channel 1/Key 40
//   PLC/PLC Instance <-> EtherCAT Master BKCUCX/TcTerminals210_EK1100_1/TcTerminals210_1BK1250/A_0007(CPx9xx-4 LEDs/Buttons)
//     PlcTask Inputs/GVL_iXlinker.EtherCAT_Master_BKCUCX.TcTerminals210_EK1100_1.TcTerminals210_1BK1250.A_0007_CPx9xx_4_LEDs_Buttons.Channel_1.Key_1 <-> Channel 1/Key 1
//     PlcTask Inputs/GVL_iXlinker.EtherCAT_Master_BKCUCX.TcTerminals210_EK1100_1.TcTerminals210_1BK1250.A_0007_CPx9xx_4_LEDs_Buttons.Channel_1.Key_2 <-> Channel 1/Key 2
//     PlcTask Inputs/GVL_iXlinker.EtherCAT_Master_BKCUCX.TcTerminals210_EK1100_1.TcTerminals210_1BK1250.A_0007_CPx9xx_4_LEDs_Buttons.Channel_1.Key_3 <-> Channel 1/Key 3
//     PlcTask Inputs/GVL_iXlinker.EtherCAT_Master_BKCUCX.TcTerminals210_EK1100_1.TcTerminals210_1BK1250.A_0007_CPx9xx_4_LEDs_Buttons.Channel_1.Key_4 <-> Channel 1/Key 4
//     PlcTask Outputs/GVL_iXlinker.EtherCAT_Master_BKCUCX.TcTerminals210_EK1100_1.TcTerminals210_1BK1250.A_0007_CPx9xx_4_LEDs_Buttons.Channel_1.LED_1 <-> Channel 1/LED 1
//     PlcTask Outputs/GVL_iXlinker.EtherCAT_Master_BKCUCX.TcTerminals210_EK1100_1.TcTerminals210_1BK1250.A_0007_CPx9xx_4_LEDs_Buttons.Channel_1.LED_2 <-> Channel 1/LED 2
//     PlcTask Outputs/GVL_iXlinker.EtherCAT_Master_BKCUCX.TcTerminals210_EK1100_1.TcTerminals210_1BK1250.A_0007_CPx9xx_4_LEDs_Buttons.Channel_1.LED_3 <-> Channel 1/LED 3
//     PlcTask Outputs/GVL_iXlinker.EtherCAT_Master_BKCUCX.TcTerminals210_EK1100_1.TcTerminals210_1BK1250.A_0007_CPx9xx_4_LEDs_Buttons.Channel_1.LED_4 <-> Channel 1/LED 4
//   PLC/PLC Instance <-> EtherCAT Master BKCUCX/TcTerminals210_EK1100_1/TcTerminals210_1BK1250/A_0008(CPx9xx-8 LEDs/Buttons)
//     PlcTask Inputs/GVL_iXlinker.EtherCAT_Master_BKCUCX.TcTerminals210_EK1100_1.TcTerminals210_1BK1250.A_0008_CPx9xx_8_LEDs_Buttons.Channel_1.Key_1 <-> Channel 1/Key 1
//     PlcTask Inputs/GVL_iXlinker.EtherCAT_Master_BKCUCX.TcTerminals210_EK1100_1.TcTerminals210_1BK1250.A_0008_CPx9xx_8_LEDs_Buttons.Channel_1.Key_2 <-> Channel 1/Key 2
//     PlcTask Inputs/GVL_iXlinker.EtherCAT_Master_BKCUCX.TcTerminals210_EK1100_1.TcTerminals210_1BK1250.A_0008_CPx9xx_8_LEDs_Buttons.Channel_1.Key_3 <-> Channel 1/Key 3
//     PlcTask Inputs/GVL_iXlinker.EtherCAT_Master_BKCUCX.TcTerminals210_EK1100_1.TcTerminals210_1BK1250.A_0008_CPx9xx_8_LEDs_Buttons.Channel_1.Key_4 <-> Channel 1/Key 4
//     PlcTask Inputs/GVL_iXlinker.EtherCAT_Master_BKCUCX.TcTerminals210_EK1100_1.TcTerminals210_1BK1250.A_0008_CPx9xx_8_LEDs_Buttons.Channel_1.Key_5 <-> Channel 1/Key 5
//     PlcTask Inputs/GVL_iXlinker.EtherCAT_Master_BKCUCX.TcTerminals210_EK1100_1.TcTerminals210_1BK1250.A_0008_CPx9xx_8_LEDs_Buttons.Channel_1.Key_6 <-> Channel 1/Key 6
//     PlcTask Inputs/GVL_iXlinker.EtherCAT_Master_BKCUCX.TcTerminals210_EK1100_1.TcTerminals210_1BK1250.A_0008_CPx9xx_8_LEDs_Buttons.Channel_1.Key_7 <-> Channel 1/Key 7
//     PlcTask Inputs/GVL_iXlinker.EtherCAT_Master_BKCUCX.TcTerminals210_EK1100_1.TcTerminals210_1BK1250.A_0008_CPx9xx_8_LEDs_Buttons.Channel_1.Key_8 <-> Channel 1/Key 8
//     PlcTask Outputs/GVL_iXlinker.EtherCAT_Master_BKCUCX.TcTerminals210_EK1100_1.TcTerminals210_1BK1250.A_0008_CPx9xx_8_LEDs_Buttons.Channel_1.LED_1 <-> Channel 1/LED 1
//     PlcTask Outputs/GVL_iXlinker.EtherCAT_Master_BKCUCX.TcTerminals210_EK1100_1.TcTerminals210_1BK1250.A_0008_CPx9xx_8_LEDs_Buttons.Channel_1.LED_2 <-> Channel 1/LED 2
//     PlcTask Outputs/GVL_iXlinker.EtherCAT_Master_BKCUCX.TcTerminals210_EK1100_1.TcTerminals210_1BK1250.A_0008_CPx9xx_8_LEDs_Buttons.Channel_1.LED_3 <-> Channel 1/LED 3
//     PlcTask Outputs/GVL_iXlinker.EtherCAT_Master_BKCUCX.TcTerminals210_EK1100_1.TcTerminals210_1BK1250.A_0008_CPx9xx_8_LEDs_Buttons.Channel_1.LED_4 <-> Channel 1/LED 4
//     PlcTask Outputs/GVL_iXlinker.EtherCAT_Master_BKCUCX.TcTerminals210_EK1100_1.TcTerminals210_1BK1250.A_0008_CPx9xx_8_LEDs_Buttons.Channel_1.LED_5 <-> Channel 1/LED 5
//     PlcTask Outputs/GVL_iXlinker.EtherCAT_Master_BKCUCX.TcTerminals210_EK1100_1.TcTerminals210_1BK1250.A_0008_CPx9xx_8_LEDs_Buttons.Channel_1.LED_6 <-> Channel 1/LED 6
//     PlcTask Outputs/GVL_iXlinker.EtherCAT_Master_BKCUCX.TcTerminals210_EK1100_1.TcTerminals210_1BK1250.A_0008_CPx9xx_8_LEDs_Buttons.Channel_1.LED_7 <-> Channel 1/LED 7
//     PlcTask Outputs/GVL_iXlinker.EtherCAT_Master_BKCUCX.TcTerminals210_EK1100_1.TcTerminals210_1BK1250.A_0008_CPx9xx_8_LEDs_Buttons.Channel_1.LED_8 <-> Channel 1/LED 8
//   PLC/PLC Instance <-> EtherCAT Master BKCUCX/TcTerminals210_EK1100_1/TcTerminals210_1BK1250/A_0009(CPx9xx-12 LEDs/Buttons)
//     PlcTask Inputs/GVL_iXlinker.EtherCAT_Master_BKCUCX.TcTerminals210_EK1100_1.TcTerminals210_1BK1250.A_0009_CPx9xx_12_LEDs_Buttons.Channel_1.Key_1 <-> Channel 1/Key 1
//     PlcTask Inputs/GVL_iXlinker.EtherCAT_Master_BKCUCX.TcTerminals210_EK1100_1.TcTerminals210_1BK1250.A_0009_CPx9xx_12_LEDs_Buttons.Channel_1.Key_2 <-> Channel 1/Key 2
//     PlcTask Inputs/GVL_iXlinker.EtherCAT_Master_BKCUCX.TcTerminals210_EK1100_1.TcTerminals210_1BK1250.A_0009_CPx9xx_12_LEDs_Buttons.Channel_1.Key_3 <-> Channel 1/Key 3
//     PlcTask Inputs/GVL_iXlinker.EtherCAT_Master_BKCUCX.TcTerminals210_EK1100_1.TcTerminals210_1BK1250.A_0009_CPx9xx_12_LEDs_Buttons.Channel_1.Key_4 <-> Channel 1/Key 4
//     PlcTask Inputs/GVL_iXlinker.EtherCAT_Master_BKCUCX.TcTerminals210_EK1100_1.TcTerminals210_1BK1250.A_0009_CPx9xx_12_LEDs_Buttons.Channel_1.Key_5 <-> Channel 1/Key 5
//     PlcTask Inputs/GVL_iXlinker.EtherCAT_Master_BKCUCX.TcTerminals210_EK1100_1.TcTerminals210_1BK1250.A_0009_CPx9xx_12_LEDs_Buttons.Channel_1.Key_6 <-> Channel 1/Key 6
//     PlcTask Inputs/GVL_iXlinker.EtherCAT_Master_BKCUCX.TcTerminals210_EK1100_1.TcTerminals210_1BK1250.A_0009_CPx9xx_12_LEDs_Buttons.Channel_1.Key_7 <-> Channel 1/Key 7
//     PlcTask Inputs/GVL_iXlinker.EtherCAT_Master_BKCUCX.TcTerminals210_EK1100_1.TcTerminals210_1BK1250.A_0009_CPx9xx_12_LEDs_Buttons.Channel_1.Key_8 <-> Channel 1/Key 8
//     PlcTask Inputs/GVL_iXlinker.EtherCAT_Master_BKCUCX.TcTerminals210_EK1100_1.TcTerminals210_1BK1250.A_0009_CPx9xx_12_LEDs_Buttons.Channel_1.Key_9 <-> Channel 1/Key 9
//     PlcTask Inputs/GVL_iXlinker.EtherCAT_Master_BKCUCX.TcTerminals210_EK1100_1.TcTerminals210_1BK1250.A_0009_CPx9xx_12_LEDs_Buttons.Channel_1.Key_10 <-> Channel 1/Key 10
//     PlcTask Inputs/GVL_iXlinker.EtherCAT_Master_BKCUCX.TcTerminals210_EK1100_1.TcTerminals210_1BK1250.A_0009_CPx9xx_12_LEDs_Buttons.Channel_1.Key_11 <-> Channel 1/Key 11
//     PlcTask Inputs/GVL_iXlinker.EtherCAT_Master_BKCUCX.TcTerminals210_EK1100_1.TcTerminals210_1BK1250.A_0009_CPx9xx_12_LEDs_Buttons.Channel_1.Key_12 <-> Channel 1/Key 12
//     PlcTask Outputs/GVL_iXlinker.EtherCAT_Master_BKCUCX.TcTerminals210_EK1100_1.TcTerminals210_1BK1250.A_0009_CPx9xx_12_LEDs_Buttons.Channel_1.LED_1 <-> Channel 1/LED 1
//     PlcTask Outputs/GVL_iXlinker.EtherCAT_Master_BKCUCX.TcTerminals210_EK1100_1.TcTerminals210_1BK1250.A_0009_CPx9xx_12_LEDs_Buttons.Channel_1.LED_2 <-> Channel 1/LED 2
//     PlcTask Outputs/GVL_iXlinker.EtherCAT_Master_BKCUCX.TcTerminals210_EK1100_1.TcTerminals210_1BK1250.A_0009_CPx9xx_12_LEDs_Buttons.Channel_1.LED_3 <-> Channel 1/LED 3
//     PlcTask Outputs/GVL_iXlinker.EtherCAT_Master_BKCUCX.TcTerminals210_EK1100_1.TcTerminals210_1BK1250.A_0009_CPx9xx_12_LEDs_Buttons.Channel_1.LED_4 <-> Channel 1/LED 4
//     PlcTask Outputs/GVL_iXlinker.EtherCAT_Master_BKCUCX.TcTerminals210_EK1100_1.TcTerminals210_1BK1250.A_0009_CPx9xx_12_LEDs_Buttons.Channel_1.LED_5 <-> Channel 1/LED 5
//     PlcTask Outputs/GVL_iXlinker.EtherCAT_Master_BKCUCX.TcTerminals210_EK1100_1.TcTerminals210_1BK1250.A_0009_CPx9xx_12_LEDs_Buttons.Channel_1.LED_6 <-> Channel 1/LED 6
//     PlcTask Outputs/GVL_iXlinker.EtherCAT_Master_BKCUCX.TcTerminals210_EK1100_1.TcTerminals210_1BK1250.A_0009_CPx9xx_12_LEDs_Buttons.Channel_1.LED_7 <-> Channel 1/LED 7
//     PlcTask Outputs/GVL_iXlinker.EtherCAT_Master_BKCUCX.TcTerminals210_EK1100_1.TcTerminals210_1BK1250.A_0009_CPx9xx_12_LEDs_Buttons.Channel_1.LED_8 <-> Channel 1/LED 8
//     PlcTask Outputs/GVL_iXlinker.EtherCAT_Master_BKCUCX.TcTerminals210_EK1100_1.TcTerminals210_1BK1250.A_0009_CPx9xx_12_LEDs_Buttons.Channel_1.LED_9 <-> Channel 1/LED 9
//     PlcTask Outputs/GVL_iXlinker.EtherCAT_Master_BKCUCX.TcTerminals210_EK1100_1.TcTerminals210_1BK1250.A_0009_CPx9xx_12_LEDs_Buttons.Channel_1.LED_10 <-> Channel 1/LED 10
//     PlcTask Outputs/GVL_iXlinker.EtherCAT_Master_BKCUCX.TcTerminals210_EK1100_1.TcTerminals210_1BK1250.A_0009_CPx9xx_12_LEDs_Buttons.Channel_1.LED_11 <-> Channel 1/LED 11
//     PlcTask Outputs/GVL_iXlinker.EtherCAT_Master_BKCUCX.TcTerminals210_EK1100_1.TcTerminals210_1BK1250.A_0009_CPx9xx_12_LEDs_Buttons.Channel_1.LED_12 <-> Channel 1/LED 12
//   PLC/PLC Instance <-> EtherCAT Master BKCUCX/TcTerminals210_EK1100_1/TcTerminals210_1BK1250/A_0010(CPx9xx-16 LEDs/Buttons)
//     PlcTask Inputs/GVL_iXlinker.EtherCAT_Master_BKCUCX.TcTerminals210_EK1100_1.TcTerminals210_1BK1250.A_0010_CPx9xx_16_LEDs_Buttons.Channel_1.Key_1 <-> Channel 1/Key 1
//     PlcTask Inputs/GVL_iXlinker.EtherCAT_Master_BKCUCX.TcTerminals210_EK1100_1.TcTerminals210_1BK1250.A_0010_CPx9xx_16_LEDs_Buttons.Channel_1.Key_2 <-> Channel 1/Key 2
//     PlcTask Inputs/GVL_iXlinker.EtherCAT_Master_BKCUCX.TcTerminals210_EK1100_1.TcTerminals210_1BK1250.A_0010_CPx9xx_16_LEDs_Buttons.Channel_1.Key_3 <-> Channel 1/Key 3
//     PlcTask Inputs/GVL_iXlinker.EtherCAT_Master_BKCUCX.TcTerminals210_EK1100_1.TcTerminals210_1BK1250.A_0010_CPx9xx_16_LEDs_Buttons.Channel_1.Key_4 <-> Channel 1/Key 4
//     PlcTask Inputs/GVL_iXlinker.EtherCAT_Master_BKCUCX.TcTerminals210_EK1100_1.TcTerminals210_1BK1250.A_0010_CPx9xx_16_LEDs_Buttons.Channel_1.Key_5 <-> Channel 1/Key 5
//     PlcTask Inputs/GVL_iXlinker.EtherCAT_Master_BKCUCX.TcTerminals210_EK1100_1.TcTerminals210_1BK1250.A_0010_CPx9xx_16_LEDs_Buttons.Channel_1.Key_6 <-> Channel 1/Key 6
//     PlcTask Inputs/GVL_iXlinker.EtherCAT_Master_BKCUCX.TcTerminals210_EK1100_1.TcTerminals210_1BK1250.A_0010_CPx9xx_16_LEDs_Buttons.Channel_1.Key_7 <-> Channel 1/Key 7
//     PlcTask Inputs/GVL_iXlinker.EtherCAT_Master_BKCUCX.TcTerminals210_EK1100_1.TcTerminals210_1BK1250.A_0010_CPx9xx_16_LEDs_Buttons.Channel_1.Key_8 <-> Channel 1/Key 8
//     PlcTask Inputs/GVL_iXlinker.EtherCAT_Master_BKCUCX.TcTerminals210_EK1100_1.TcTerminals210_1BK1250.A_0010_CPx9xx_16_LEDs_Buttons.Channel_1.Key_9 <-> Channel 1/Key 9
//     PlcTask Inputs/GVL_iXlinker.EtherCAT_Master_BKCUCX.TcTerminals210_EK1100_1.TcTerminals210_1BK1250.A_0010_CPx9xx_16_LEDs_Buttons.Channel_1.Key_10 <-> Channel 1/Key 10
//     PlcTask Inputs/GVL_iXlinker.EtherCAT_Master_BKCUCX.TcTerminals210_EK1100_1.TcTerminals210_1BK1250.A_0010_CPx9xx_16_LEDs_Buttons.Channel_1.Key_11 <-> Channel 1/Key 11
//     PlcTask Inputs/GVL_iXlinker.EtherCAT_Master_BKCUCX.TcTerminals210_EK1100_1.TcTerminals210_1BK1250.A_0010_CPx9xx_16_LEDs_Buttons.Channel_1.Key_12 <-> Channel 1/Key 12
//     PlcTask Inputs/GVL_iXlinker.EtherCAT_Master_BKCUCX.TcTerminals210_EK1100_1.TcTerminals210_1BK1250.A_0010_CPx9xx_16_LEDs_Buttons.Channel_1.Key_13 <-> Channel 1/Key 13
//     PlcTask Inputs/GVL_iXlinker.EtherCAT_Master_BKCUCX.TcTerminals210_EK1100_1.TcTerminals210_1BK1250.A_0010_CPx9xx_16_LEDs_Buttons.Channel_1.Key_14 <-> Channel 1/Key 14
//     PlcTask Inputs/GVL_iXlinker.EtherCAT_Master_BKCUCX.TcTerminals210_EK1100_1.TcTerminals210_1BK1250.A_0010_CPx9xx_16_LEDs_Buttons.Channel_1.Key_15 <-> Channel 1/Key 15
//     PlcTask Inputs/GVL_iXlinker.EtherCAT_Master_BKCUCX.TcTerminals210_EK1100_1.TcTerminals210_1BK1250.A_0010_CPx9xx_16_LEDs_Buttons.Channel_1.Key_16 <-> Channel 1/Key 16
//     PlcTask Outputs/GVL_iXlinker.EtherCAT_Master_BKCUCX.TcTerminals210_EK1100_1.TcTerminals210_1BK1250.A_0010_CPx9xx_16_LEDs_Buttons.Channel_1.LED_1 <-> Channel 1/LED 1
//     PlcTask Outputs/GVL_iXlinker.EtherCAT_Master_BKCUCX.TcTerminals210_EK1100_1.TcTerminals210_1BK1250.A_0010_CPx9xx_16_LEDs_Buttons.Channel_1.LED_2 <-> Channel 1/LED 2
//     PlcTask Outputs/GVL_iXlinker.EtherCAT_Master_BKCUCX.TcTerminals210_EK1100_1.TcTerminals210_1BK1250.A_0010_CPx9xx_16_LEDs_Buttons.Channel_1.LED_3 <-> Channel 1/LED 3
//     PlcTask Outputs/GVL_iXlinker.EtherCAT_Master_BKCUCX.TcTerminals210_EK1100_1.TcTerminals210_1BK1250.A_0010_CPx9xx_16_LEDs_Buttons.Channel_1.LED_4 <-> Channel 1/LED 4
//     PlcTask Outputs/GVL_iXlinker.EtherCAT_Master_BKCUCX.TcTerminals210_EK1100_1.TcTerminals210_1BK1250.A_0010_CPx9xx_16_LEDs_Buttons.Channel_1.LED_5 <-> Channel 1/LED 5
//     PlcTask Outputs/GVL_iXlinker.EtherCAT_Master_BKCUCX.TcTerminals210_EK1100_1.TcTerminals210_1BK1250.A_0010_CPx9xx_16_LEDs_Buttons.Channel_1.LED_6 <-> Channel 1/LED 6
//     PlcTask Outputs/GVL_iXlinker.EtherCAT_Master_BKCUCX.TcTerminals210_EK1100_1.TcTerminals210_1BK1250.A_0010_CPx9xx_16_LEDs_Buttons.Channel_1.LED_7 <-> Channel 1/LED 7
//     PlcTask Outputs/GVL_iXlinker.EtherCAT_Master_BKCUCX.TcTerminals210_EK1100_1.TcTerminals210_1BK1250.A_0010_CPx9xx_16_LEDs_Buttons.Channel_1.LED_8 <-> Channel 1/LED 8
//     PlcTask Outputs/GVL_iXlinker.EtherCAT_Master_BKCUCX.TcTerminals210_EK1100_1.TcTerminals210_1BK1250.A_0010_CPx9xx_16_LEDs_Buttons.Channel_1.LED_9 <-> Channel 1/LED 9
//     PlcTask Outputs/GVL_iXlinker.EtherCAT_Master_BKCUCX.TcTerminals210_EK1100_1.TcTerminals210_1BK1250.A_0010_CPx9xx_16_LEDs_Buttons.Channel_1.LED_10 <-> Channel 1/LED 10
//     PlcTask Outputs/GVL_iXlinker.EtherCAT_Master_BKCUCX.TcTerminals210_EK1100_1.TcTerminals210_1BK1250.A_0010_CPx9xx_16_LEDs_Buttons.Channel_1.LED_11 <-> Channel 1/LED 11
//     PlcTask Outputs/GVL_iXlinker.EtherCAT_Master_BKCUCX.TcTerminals210_EK1100_1.TcTerminals210_1BK1250.A_0010_CPx9xx_16_LEDs_Buttons.Channel_1.LED_12 <-> Channel 1/LED 12
//     PlcTask Outputs/GVL_iXlinker.EtherCAT_Master_BKCUCX.TcTerminals210_EK1100_1.TcTerminals210_1BK1250.A_0010_CPx9xx_16_LEDs_Buttons.Channel_1.LED_13 <-> Channel 1/LED 13
//     PlcTask Outputs/GVL_iXlinker.EtherCAT_Master_BKCUCX.TcTerminals210_EK1100_1.TcTerminals210_1BK1250.A_0010_CPx9xx_16_LEDs_Buttons.Channel_1.LED_14 <-> Channel 1/LED 14
//     PlcTask Outputs/GVL_iXlinker.EtherCAT_Master_BKCUCX.TcTerminals210_EK1100_1.TcTerminals210_1BK1250.A_0010_CPx9xx_16_LEDs_Buttons.Channel_1.LED_15 <-> Channel 1/LED 15
//     PlcTask Outputs/GVL_iXlinker.EtherCAT_Master_BKCUCX.TcTerminals210_EK1100_1.TcTerminals210_1BK1250.A_0010_CPx9xx_16_LEDs_Buttons.Channel_1.LED_16 <-> Channel 1/LED 16
//   PLC/PLC Instance <-> EtherCAT Master BKCUCX/TcTerminals210_EK1100_1/TcTerminals210_1BK1250/A_0011(CPx9xx-20 LEDs/Buttons)
//     PlcTask Inputs/GVL_iXlinker.EtherCAT_Master_BKCUCX.TcTerminals210_EK1100_1.TcTerminals210_1BK1250.A_0011_CPx9xx_20_LEDs_Buttons.Channel_1.Key_1 <-> Channel 1/Key 1
//     PlcTask Inputs/GVL_iXlinker.EtherCAT_Master_BKCUCX.TcTerminals210_EK1100_1.TcTerminals210_1BK1250.A_0011_CPx9xx_20_LEDs_Buttons.Channel_1.Key_2 <-> Channel 1/Key 2
//     PlcTask Inputs/GVL_iXlinker.EtherCAT_Master_BKCUCX.TcTerminals210_EK1100_1.TcTerminals210_1BK1250.A_0011_CPx9xx_20_LEDs_Buttons.Channel_1.Key_3 <-> Channel 1/Key 3
//     PlcTask Inputs/GVL_iXlinker.EtherCAT_Master_BKCUCX.TcTerminals210_EK1100_1.TcTerminals210_1BK1250.A_0011_CPx9xx_20_LEDs_Buttons.Channel_1.Key_4 <-> Channel 1/Key 4
//     PlcTask Inputs/GVL_iXlinker.EtherCAT_Master_BKCUCX.TcTerminals210_EK1100_1.TcTerminals210_1BK1250.A_0011_CPx9xx_20_LEDs_Buttons.Channel_1.Key_5 <-> Channel 1/Key 5
//     PlcTask Inputs/GVL_iXlinker.EtherCAT_Master_BKCUCX.TcTerminals210_EK1100_1.TcTerminals210_1BK1250.A_0011_CPx9xx_20_LEDs_Buttons.Channel_1.Key_6 <-> Channel 1/Key 6
//     PlcTask Inputs/GVL_iXlinker.EtherCAT_Master_BKCUCX.TcTerminals210_EK1100_1.TcTerminals210_1BK1250.A_0011_CPx9xx_20_LEDs_Buttons.Channel_1.Key_7 <-> Channel 1/Key 7
//     PlcTask Inputs/GVL_iXlinker.EtherCAT_Master_BKCUCX.TcTerminals210_EK1100_1.TcTerminals210_1BK1250.A_0011_CPx9xx_20_LEDs_Buttons.Channel_1.Key_8 <-> Channel 1/Key 8
//     PlcTask Inputs/GVL_iXlinker.EtherCAT_Master_BKCUCX.TcTerminals210_EK1100_1.TcTerminals210_1BK1250.A_0011_CPx9xx_20_LEDs_Buttons.Channel_1.Key_9 <-> Channel 1/Key 9
//     PlcTask Inputs/GVL_iXlinker.EtherCAT_Master_BKCUCX.TcTerminals210_EK1100_1.TcTerminals210_1BK1250.A_0011_CPx9xx_20_LEDs_Buttons.Channel_1.Key_10 <-> Channel 1/Key 10
//     PlcTask Inputs/GVL_iXlinker.EtherCAT_Master_BKCUCX.TcTerminals210_EK1100_1.TcTerminals210_1BK1250.A_0011_CPx9xx_20_LEDs_Buttons.Channel_1.Key_11 <-> Channel 1/Key 11
//     PlcTask Inputs/GVL_iXlinker.EtherCAT_Master_BKCUCX.TcTerminals210_EK1100_1.TcTerminals210_1BK1250.A_0011_CPx9xx_20_LEDs_Buttons.Channel_1.Key_12 <-> Channel 1/Key 12
//     PlcTask Inputs/GVL_iXlinker.EtherCAT_Master_BKCUCX.TcTerminals210_EK1100_1.TcTerminals210_1BK1250.A_0011_CPx9xx_20_LEDs_Buttons.Channel_1.Key_13 <-> Channel 1/Key 13
//     PlcTask Inputs/GVL_iXlinker.EtherCAT_Master_BKCUCX.TcTerminals210_EK1100_1.TcTerminals210_1BK1250.A_0011_CPx9xx_20_LEDs_Buttons.Channel_1.Key_14 <-> Channel 1/Key 14
//     PlcTask Inputs/GVL_iXlinker.EtherCAT_Master_BKCUCX.TcTerminals210_EK1100_1.TcTerminals210_1BK1250.A_0011_CPx9xx_20_LEDs_Buttons.Channel_1.Key_15 <-> Channel 1/Key 15
//     PlcTask Inputs/GVL_iXlinker.EtherCAT_Master_BKCUCX.TcTerminals210_EK1100_1.TcTerminals210_1BK1250.A_0011_CPx9xx_20_LEDs_Buttons.Channel_1.Key_16 <-> Channel 1/Key 16
//     PlcTask Inputs/GVL_iXlinker.EtherCAT_Master_BKCUCX.TcTerminals210_EK1100_1.TcTerminals210_1BK1250.A_0011_CPx9xx_20_LEDs_Buttons.Channel_1.Key_17 <-> Channel 1/Key 17
//     PlcTask Inputs/GVL_iXlinker.EtherCAT_Master_BKCUCX.TcTerminals210_EK1100_1.TcTerminals210_1BK1250.A_0011_CPx9xx_20_LEDs_Buttons.Channel_1.Key_18 <-> Channel 1/Key 18
//     PlcTask Inputs/GVL_iXlinker.EtherCAT_Master_BKCUCX.TcTerminals210_EK1100_1.TcTerminals210_1BK1250.A_0011_CPx9xx_20_LEDs_Buttons.Channel_1.Key_19 <-> Channel 1/Key 19
//     PlcTask Inputs/GVL_iXlinker.EtherCAT_Master_BKCUCX.TcTerminals210_EK1100_1.TcTerminals210_1BK1250.A_0011_CPx9xx_20_LEDs_Buttons.Channel_1.Key_20 <-> Channel 1/Key 20
//     PlcTask Outputs/GVL_iXlinker.EtherCAT_Master_BKCUCX.TcTerminals210_EK1100_1.TcTerminals210_1BK1250.A_0011_CPx9xx_20_LEDs_Buttons.Channel_1.LED_1 <-> Channel 1/LED 1
//     PlcTask Outputs/GVL_iXlinker.EtherCAT_Master_BKCUCX.TcTerminals210_EK1100_1.TcTerminals210_1BK1250.A_0011_CPx9xx_20_LEDs_Buttons.Channel_1.LED_2 <-> Channel 1/LED 2
//     PlcTask Outputs/GVL_iXlinker.EtherCAT_Master_BKCUCX.TcTerminals210_EK1100_1.TcTerminals210_1BK1250.A_0011_CPx9xx_20_LEDs_Buttons.Channel_1.LED_3 <-> Channel 1/LED 3
//     PlcTask Outputs/GVL_iXlinker.EtherCAT_Master_BKCUCX.TcTerminals210_EK1100_1.TcTerminals210_1BK1250.A_0011_CPx9xx_20_LEDs_Buttons.Channel_1.LED_4 <-> Channel 1/LED 4
//     PlcTask Outputs/GVL_iXlinker.EtherCAT_Master_BKCUCX.TcTerminals210_EK1100_1.TcTerminals210_1BK1250.A_0011_CPx9xx_20_LEDs_Buttons.Channel_1.LED_5 <-> Channel 1/LED 5
//     PlcTask Outputs/GVL_iXlinker.EtherCAT_Master_BKCUCX.TcTerminals210_EK1100_1.TcTerminals210_1BK1250.A_0011_CPx9xx_20_LEDs_Buttons.Channel_1.LED_6 <-> Channel 1/LED 6
//     PlcTask Outputs/GVL_iXlinker.EtherCAT_Master_BKCUCX.TcTerminals210_EK1100_1.TcTerminals210_1BK1250.A_0011_CPx9xx_20_LEDs_Buttons.Channel_1.LED_7 <-> Channel 1/LED 7
//     PlcTask Outputs/GVL_iXlinker.EtherCAT_Master_BKCUCX.TcTerminals210_EK1100_1.TcTerminals210_1BK1250.A_0011_CPx9xx_20_LEDs_Buttons.Channel_1.LED_8 <-> Channel 1/LED 8
//     PlcTask Outputs/GVL_iXlinker.EtherCAT_Master_BKCUCX.TcTerminals210_EK1100_1.TcTerminals210_1BK1250.A_0011_CPx9xx_20_LEDs_Buttons.Channel_1.LED_9 <-> Channel 1/LED 9
//     PlcTask Outputs/GVL_iXlinker.EtherCAT_Master_BKCUCX.TcTerminals210_EK1100_1.TcTerminals210_1BK1250.A_0011_CPx9xx_20_LEDs_Buttons.Channel_1.LED_10 <-> Channel 1/LED 10
//     PlcTask Outputs/GVL_iXlinker.EtherCAT_Master_BKCUCX.TcTerminals210_EK1100_1.TcTerminals210_1BK1250.A_0011_CPx9xx_20_LEDs_Buttons.Channel_1.LED_11 <-> Channel 1/LED 11
//     PlcTask Outputs/GVL_iXlinker.EtherCAT_Master_BKCUCX.TcTerminals210_EK1100_1.TcTerminals210_1BK1250.A_0011_CPx9xx_20_LEDs_Buttons.Channel_1.LED_12 <-> Channel 1/LED 12
//     PlcTask Outputs/GVL_iXlinker.EtherCAT_Master_BKCUCX.TcTerminals210_EK1100_1.TcTerminals210_1BK1250.A_0011_CPx9xx_20_LEDs_Buttons.Channel_1.LED_13 <-> Channel 1/LED 13
//     PlcTask Outputs/GVL_iXlinker.EtherCAT_Master_BKCUCX.TcTerminals210_EK1100_1.TcTerminals210_1BK1250.A_0011_CPx9xx_20_LEDs_Buttons.Channel_1.LED_14 <-> Channel 1/LED 14
//     PlcTask Outputs/GVL_iXlinker.EtherCAT_Master_BKCUCX.TcTerminals210_EK1100_1.TcTerminals210_1BK1250.A_0011_CPx9xx_20_LEDs_Buttons.Channel_1.LED_15 <-> Channel 1/LED 15
//     PlcTask Outputs/GVL_iXlinker.EtherCAT_Master_BKCUCX.TcTerminals210_EK1100_1.TcTerminals210_1BK1250.A_0011_CPx9xx_20_LEDs_Buttons.Channel_1.LED_16 <-> Channel 1/LED 16
//     PlcTask Outputs/GVL_iXlinker.EtherCAT_Master_BKCUCX.TcTerminals210_EK1100_1.TcTerminals210_1BK1250.A_0011_CPx9xx_20_LEDs_Buttons.Channel_1.LED_17 <-> Channel 1/LED 17
//     PlcTask Outputs/GVL_iXlinker.EtherCAT_Master_BKCUCX.TcTerminals210_EK1100_1.TcTerminals210_1BK1250.A_0011_CPx9xx_20_LEDs_Buttons.Channel_1.LED_18 <-> Channel 1/LED 18
//     PlcTask Outputs/GVL_iXlinker.EtherCAT_Master_BKCUCX.TcTerminals210_EK1100_1.TcTerminals210_1BK1250.A_0011_CPx9xx_20_LEDs_Buttons.Channel_1.LED_19 <-> Channel 1/LED 19
//     PlcTask Outputs/GVL_iXlinker.EtherCAT_Master_BKCUCX.TcTerminals210_EK1100_1.TcTerminals210_1BK1250.A_0011_CPx9xx_20_LEDs_Buttons.Channel_1.LED_20 <-> Channel 1/LED 20
//   PLC/PLC Instance <-> EtherCAT Master BKCUCX/TcTerminals210_EK1100_1/TcTerminals210_1BK1250/A_0012(CPx9xx-24 LEDs/Buttons)
//     PlcTask Inputs/GVL_iXlinker.EtherCAT_Master_BKCUCX.TcTerminals210_EK1100_1.TcTerminals210_1BK1250.A_0012_CPx9xx_24_LEDs_Buttons.Channel_1.Key_1 <-> Channel 1/Key 1
//     PlcTask Inputs/GVL_iXlinker.EtherCAT_Master_BKCUCX.TcTerminals210_EK1100_1.TcTerminals210_1BK1250.A_0012_CPx9xx_24_LEDs_Buttons.Channel_1.Key_2 <-> Channel 1/Key 2
//     PlcTask Inputs/GVL_iXlinker.EtherCAT_Master_BKCUCX.TcTerminals210_EK1100_1.TcTerminals210_1BK1250.A_0012_CPx9xx_24_LEDs_Buttons.Channel_1.Key_3 <-> Channel 1/Key 3
//     PlcTask Inputs/GVL_iXlinker.EtherCAT_Master_BKCUCX.TcTerminals210_EK1100_1.TcTerminals210_1BK1250.A_0012_CPx9xx_24_LEDs_Buttons.Channel_1.Key_4 <-> Channel 1/Key 4
//     PlcTask Inputs/GVL_iXlinker.EtherCAT_Master_BKCUCX.TcTerminals210_EK1100_1.TcTerminals210_1BK1250.A_0012_CPx9xx_24_LEDs_Buttons.Channel_1.Key_5 <-> Channel 1/Key 5
//     PlcTask Inputs/GVL_iXlinker.EtherCAT_Master_BKCUCX.TcTerminals210_EK1100_1.TcTerminals210_1BK1250.A_0012_CPx9xx_24_LEDs_Buttons.Channel_1.Key_6 <-> Channel 1/Key 6
//     PlcTask Inputs/GVL_iXlinker.EtherCAT_Master_BKCUCX.TcTerminals210_EK1100_1.TcTerminals210_1BK1250.A_0012_CPx9xx_24_LEDs_Buttons.Channel_1.Key_7 <-> Channel 1/Key 7
//     PlcTask Inputs/GVL_iXlinker.EtherCAT_Master_BKCUCX.TcTerminals210_EK1100_1.TcTerminals210_1BK1250.A_0012_CPx9xx_24_LEDs_Buttons.Channel_1.Key_8 <-> Channel 1/Key 8
//     PlcTask Inputs/GVL_iXlinker.EtherCAT_Master_BKCUCX.TcTerminals210_EK1100_1.TcTerminals210_1BK1250.A_0012_CPx9xx_24_LEDs_Buttons.Channel_1.Key_9 <-> Channel 1/Key 9
//     PlcTask Inputs/GVL_iXlinker.EtherCAT_Master_BKCUCX.TcTerminals210_EK1100_1.TcTerminals210_1BK1250.A_0012_CPx9xx_24_LEDs_Buttons.Channel_1.Key_10 <-> Channel 1/Key 10
//     PlcTask Inputs/GVL_iXlinker.EtherCAT_Master_BKCUCX.TcTerminals210_EK1100_1.TcTerminals210_1BK1250.A_0012_CPx9xx_24_LEDs_Buttons.Channel_1.Key_11 <-> Channel 1/Key 11
//     PlcTask Inputs/GVL_iXlinker.EtherCAT_Master_BKCUCX.TcTerminals210_EK1100_1.TcTerminals210_1BK1250.A_0012_CPx9xx_24_LEDs_Buttons.Channel_1.Key_12 <-> Channel 1/Key 12
//     PlcTask Inputs/GVL_iXlinker.EtherCAT_Master_BKCUCX.TcTerminals210_EK1100_1.TcTerminals210_1BK1250.A_0012_CPx9xx_24_LEDs_Buttons.Channel_1.Key_13 <-> Channel 1/Key 13
//     PlcTask Inputs/GVL_iXlinker.EtherCAT_Master_BKCUCX.TcTerminals210_EK1100_1.TcTerminals210_1BK1250.A_0012_CPx9xx_24_LEDs_Buttons.Channel_1.Key_14 <-> Channel 1/Key 14
//     PlcTask Inputs/GVL_iXlinker.EtherCAT_Master_BKCUCX.TcTerminals210_EK1100_1.TcTerminals210_1BK1250.A_0012_CPx9xx_24_LEDs_Buttons.Channel_1.Key_15 <-> Channel 1/Key 15
//     PlcTask Inputs/GVL_iXlinker.EtherCAT_Master_BKCUCX.TcTerminals210_EK1100_1.TcTerminals210_1BK1250.A_0012_CPx9xx_24_LEDs_Buttons.Channel_1.Key_16 <-> Channel 1/Key 16
//     PlcTask Inputs/GVL_iXlinker.EtherCAT_Master_BKCUCX.TcTerminals210_EK1100_1.TcTerminals210_1BK1250.A_0012_CPx9xx_24_LEDs_Buttons.Channel_1.Key_17 <-> Channel 1/Key 17
//     PlcTask Inputs/GVL_iXlinker.EtherCAT_Master_BKCUCX.TcTerminals210_EK1100_1.TcTerminals210_1BK1250.A_0012_CPx9xx_24_LEDs_Buttons.Channel_1.Key_18 <-> Channel 1/Key 18
//     PlcTask Inputs/GVL_iXlinker.EtherCAT_Master_BKCUCX.TcTerminals210_EK1100_1.TcTerminals210_1BK1250.A_0012_CPx9xx_24_LEDs_Buttons.Channel_1.Key_19 <-> Channel 1/Key 19
//     PlcTask Inputs/GVL_iXlinker.EtherCAT_Master_BKCUCX.TcTerminals210_EK1100_1.TcTerminals210_1BK1250.A_0012_CPx9xx_24_LEDs_Buttons.Channel_1.Key_20 <-> Channel 1/Key 20
//     PlcTask Inputs/GVL_iXlinker.EtherCAT_Master_BKCUCX.TcTerminals210_EK1100_1.TcTerminals210_1BK1250.A_0012_CPx9xx_24_LEDs_Buttons.Channel_1.Key_21 <-> Channel 1/Key 21
//     PlcTask Inputs/GVL_iXlinker.EtherCAT_Master_BKCUCX.TcTerminals210_EK1100_1.TcTerminals210_1BK1250.A_0012_CPx9xx_24_LEDs_Buttons.Channel_1.Key_22 <-> Channel 1/Key 22
//     PlcTask Inputs/GVL_iXlinker.EtherCAT_Master_BKCUCX.TcTerminals210_EK1100_1.TcTerminals210_1BK1250.A_0012_CPx9xx_24_LEDs_Buttons.Channel_1.Key_23 <-> Channel 1/Key 23
//     PlcTask Inputs/GVL_iXlinker.EtherCAT_Master_BKCUCX.TcTerminals210_EK1100_1.TcTerminals210_1BK1250.A_0012_CPx9xx_24_LEDs_Buttons.Channel_1.Key_24 <-> Channel 1/Key 24
//     PlcTask Outputs/GVL_iXlinker.EtherCAT_Master_BKCUCX.TcTerminals210_EK1100_1.TcTerminals210_1BK1250.A_0012_CPx9xx_24_LEDs_Buttons.Channel_1.LED_1 <-> Channel 1/LED 1
//     PlcTask Outputs/GVL_iXlinker.EtherCAT_Master_BKCUCX.TcTerminals210_EK1100_1.TcTerminals210_1BK1250.A_0012_CPx9xx_24_LEDs_Buttons.Channel_1.LED_2 <-> Channel 1/LED 2
//     PlcTask Outputs/GVL_iXlinker.EtherCAT_Master_BKCUCX.TcTerminals210_EK1100_1.TcTerminals210_1BK1250.A_0012_CPx9xx_24_LEDs_Buttons.Channel_1.LED_3 <-> Channel 1/LED 3
//     PlcTask Outputs/GVL_iXlinker.EtherCAT_Master_BKCUCX.TcTerminals210_EK1100_1.TcTerminals210_1BK1250.A_0012_CPx9xx_24_LEDs_Buttons.Channel_1.LED_4 <-> Channel 1/LED 4
//     PlcTask Outputs/GVL_iXlinker.EtherCAT_Master_BKCUCX.TcTerminals210_EK1100_1.TcTerminals210_1BK1250.A_0012_CPx9xx_24_LEDs_Buttons.Channel_1.LED_5 <-> Channel 1/LED 5
//     PlcTask Outputs/GVL_iXlinker.EtherCAT_Master_BKCUCX.TcTerminals210_EK1100_1.TcTerminals210_1BK1250.A_0012_CPx9xx_24_LEDs_Buttons.Channel_1.LED_6 <-> Channel 1/LED 6
//     PlcTask Outputs/GVL_iXlinker.EtherCAT_Master_BKCUCX.TcTerminals210_EK1100_1.TcTerminals210_1BK1250.A_0012_CPx9xx_24_LEDs_Buttons.Channel_1.LED_7 <-> Channel 1/LED 7
//     PlcTask Outputs/GVL_iXlinker.EtherCAT_Master_BKCUCX.TcTerminals210_EK1100_1.TcTerminals210_1BK1250.A_0012_CPx9xx_24_LEDs_Buttons.Channel_1.LED_8 <-> Channel 1/LED 8
//     PlcTask Outputs/GVL_iXlinker.EtherCAT_Master_BKCUCX.TcTerminals210_EK1100_1.TcTerminals210_1BK1250.A_0012_CPx9xx_24_LEDs_Buttons.Channel_1.LED_9 <-> Channel 1/LED 9
//     PlcTask Outputs/GVL_iXlinker.EtherCAT_Master_BKCUCX.TcTerminals210_EK1100_1.TcTerminals210_1BK1250.A_0012_CPx9xx_24_LEDs_Buttons.Channel_1.LED_10 <-> Channel 1/LED 10
//     PlcTask Outputs/GVL_iXlinker.EtherCAT_Master_BKCUCX.TcTerminals210_EK1100_1.TcTerminals210_1BK1250.A_0012_CPx9xx_24_LEDs_Buttons.Channel_1.LED_11 <-> Channel 1/LED 11
//     PlcTask Outputs/GVL_iXlinker.EtherCAT_Master_BKCUCX.TcTerminals210_EK1100_1.TcTerminals210_1BK1250.A_0012_CPx9xx_24_LEDs_Buttons.Channel_1.LED_12 <-> Channel 1/LED 12
//     PlcTask Outputs/GVL_iXlinker.EtherCAT_Master_BKCUCX.TcTerminals210_EK1100_1.TcTerminals210_1BK1250.A_0012_CPx9xx_24_LEDs_Buttons.Channel_1.LED_13 <-> Channel 1/LED 13
//     PlcTask Outputs/GVL_iXlinker.EtherCAT_Master_BKCUCX.TcTerminals210_EK1100_1.TcTerminals210_1BK1250.A_0012_CPx9xx_24_LEDs_Buttons.Channel_1.LED_14 <-> Channel 1/LED 14
//     PlcTask Outputs/GVL_iXlinker.EtherCAT_Master_BKCUCX.TcTerminals210_EK1100_1.TcTerminals210_1BK1250.A_0012_CPx9xx_24_LEDs_Buttons.Channel_1.LED_15 <-> Channel 1/LED 15
//     PlcTask Outputs/GVL_iXlinker.EtherCAT_Master_BKCUCX.TcTerminals210_EK1100_1.TcTerminals210_1BK1250.A_0012_CPx9xx_24_LEDs_Buttons.Channel_1.LED_16 <-> Channel 1/LED 16
//     PlcTask Outputs/GVL_iXlinker.EtherCAT_Master_BKCUCX.TcTerminals210_EK1100_1.TcTerminals210_1BK1250.A_0012_CPx9xx_24_LEDs_Buttons.Channel_1.LED_17 <-> Channel 1/LED 17
//     PlcTask Outputs/GVL_iXlinker.EtherCAT_Master_BKCUCX.TcTerminals210_EK1100_1.TcTerminals210_1BK1250.A_0012_CPx9xx_24_LEDs_Buttons.Channel_1.LED_18 <-> Channel 1/LED 18
//     PlcTask Outputs/GVL_iXlinker.EtherCAT_Master_BKCUCX.TcTerminals210_EK1100_1.TcTerminals210_1BK1250.A_0012_CPx9xx_24_LEDs_Buttons.Channel_1.LED_19 <-> Channel 1/LED 19
//     PlcTask Outputs/GVL_iXlinker.EtherCAT_Master_BKCUCX.TcTerminals210_EK1100_1.TcTerminals210_1BK1250.A_0012_CPx9xx_24_LEDs_Buttons.Channel_1.LED_20 <-> Channel 1/LED 20
//     PlcTask Outputs/GVL_iXlinker.EtherCAT_Master_BKCUCX.TcTerminals210_EK1100_1.TcTerminals210_1BK1250.A_0012_CPx9xx_24_LEDs_Buttons.Channel_1.LED_21 <-> Channel 1/LED 21
//     PlcTask Outputs/GVL_iXlinker.EtherCAT_Master_BKCUCX.TcTerminals210_EK1100_1.TcTerminals210_1BK1250.A_0012_CPx9xx_24_LEDs_Buttons.Channel_1.LED_22 <-> Channel 1/LED 22
//     PlcTask Outputs/GVL_iXlinker.EtherCAT_Master_BKCUCX.TcTerminals210_EK1100_1.TcTerminals210_1BK1250.A_0012_CPx9xx_24_LEDs_Buttons.Channel_1.LED_23 <-> Channel 1/LED 23
//     PlcTask Outputs/GVL_iXlinker.EtherCAT_Master_BKCUCX.TcTerminals210_EK1100_1.TcTerminals210_1BK1250.A_0012_CPx9xx_24_LEDs_Buttons.Channel_1.LED_24 <-> Channel 1/LED 24
//   PLC/PLC Instance <-> EtherCAT Master BKCUCX/TcTerminals210_EK1100_1/TcTerminals210_1BK1250/A_0013(CPx9xx-28 LEDs/Buttons)
//     PlcTask Inputs/GVL_iXlinker.EtherCAT_Master_BKCUCX.TcTerminals210_EK1100_1.TcTerminals210_1BK1250.A_0013_CPx9xx_28_LEDs_Buttons.Channel_1.Key_1 <-> Channel 1/Key 1
//     PlcTask Inputs/GVL_iXlinker.EtherCAT_Master_BKCUCX.TcTerminals210_EK1100_1.TcTerminals210_1BK1250.A_0013_CPx9xx_28_LEDs_Buttons.Channel_1.Key_2 <-> Channel 1/Key 2
//     PlcTask Inputs/GVL_iXlinker.EtherCAT_Master_BKCUCX.TcTerminals210_EK1100_1.TcTerminals210_1BK1250.A_0013_CPx9xx_28_LEDs_Buttons.Channel_1.Key_3 <-> Channel 1/Key 3
//     PlcTask Inputs/GVL_iXlinker.EtherCAT_Master_BKCUCX.TcTerminals210_EK1100_1.TcTerminals210_1BK1250.A_0013_CPx9xx_28_LEDs_Buttons.Channel_1.Key_4 <-> Channel 1/Key 4
//     PlcTask Inputs/GVL_iXlinker.EtherCAT_Master_BKCUCX.TcTerminals210_EK1100_1.TcTerminals210_1BK1250.A_0013_CPx9xx_28_LEDs_Buttons.Channel_1.Key_5 <-> Channel 1/Key 5
//     PlcTask Inputs/GVL_iXlinker.EtherCAT_Master_BKCUCX.TcTerminals210_EK1100_1.TcTerminals210_1BK1250.A_0013_CPx9xx_28_LEDs_Buttons.Channel_1.Key_6 <-> Channel 1/Key 6
//     PlcTask Inputs/GVL_iXlinker.EtherCAT_Master_BKCUCX.TcTerminals210_EK1100_1.TcTerminals210_1BK1250.A_0013_CPx9xx_28_LEDs_Buttons.Channel_1.Key_7 <-> Channel 1/Key 7
//     PlcTask Inputs/GVL_iXlinker.EtherCAT_Master_BKCUCX.TcTerminals210_EK1100_1.TcTerminals210_1BK1250.A_0013_CPx9xx_28_LEDs_Buttons.Channel_1.Key_8 <-> Channel 1/Key 8
//     PlcTask Inputs/GVL_iXlinker.EtherCAT_Master_BKCUCX.TcTerminals210_EK1100_1.TcTerminals210_1BK1250.A_0013_CPx9xx_28_LEDs_Buttons.Channel_1.Key_9 <-> Channel 1/Key 9
//     PlcTask Inputs/GVL_iXlinker.EtherCAT_Master_BKCUCX.TcTerminals210_EK1100_1.TcTerminals210_1BK1250.A_0013_CPx9xx_28_LEDs_Buttons.Channel_1.Key_10 <-> Channel 1/Key 10
//     PlcTask Inputs/GVL_iXlinker.EtherCAT_Master_BKCUCX.TcTerminals210_EK1100_1.TcTerminals210_1BK1250.A_0013_CPx9xx_28_LEDs_Buttons.Channel_1.Key_11 <-> Channel 1/Key 11
//     PlcTask Inputs/GVL_iXlinker.EtherCAT_Master_BKCUCX.TcTerminals210_EK1100_1.TcTerminals210_1BK1250.A_0013_CPx9xx_28_LEDs_Buttons.Channel_1.Key_12 <-> Channel 1/Key 12
//     PlcTask Inputs/GVL_iXlinker.EtherCAT_Master_BKCUCX.TcTerminals210_EK1100_1.TcTerminals210_1BK1250.A_0013_CPx9xx_28_LEDs_Buttons.Channel_1.Key_13 <-> Channel 1/Key 13
//     PlcTask Inputs/GVL_iXlinker.EtherCAT_Master_BKCUCX.TcTerminals210_EK1100_1.TcTerminals210_1BK1250.A_0013_CPx9xx_28_LEDs_Buttons.Channel_1.Key_14 <-> Channel 1/Key 14
//     PlcTask Inputs/GVL_iXlinker.EtherCAT_Master_BKCUCX.TcTerminals210_EK1100_1.TcTerminals210_1BK1250.A_0013_CPx9xx_28_LEDs_Buttons.Channel_1.Key_15 <-> Channel 1/Key 15
//     PlcTask Inputs/GVL_iXlinker.EtherCAT_Master_BKCUCX.TcTerminals210_EK1100_1.TcTerminals210_1BK1250.A_0013_CPx9xx_28_LEDs_Buttons.Channel_1.Key_16 <-> Channel 1/Key 16
//     PlcTask Inputs/GVL_iXlinker.EtherCAT_Master_BKCUCX.TcTerminals210_EK1100_1.TcTerminals210_1BK1250.A_0013_CPx9xx_28_LEDs_Buttons.Channel_1.Key_17 <-> Channel 1/Key 17
//     PlcTask Inputs/GVL_iXlinker.EtherCAT_Master_BKCUCX.TcTerminals210_EK1100_1.TcTerminals210_1BK1250.A_0013_CPx9xx_28_LEDs_Buttons.Channel_1.Key_18 <-> Channel 1/Key 18
//     PlcTask Inputs/GVL_iXlinker.EtherCAT_Master_BKCUCX.TcTerminals210_EK1100_1.TcTerminals210_1BK1250.A_0013_CPx9xx_28_LEDs_Buttons.Channel_1.Key_19 <-> Channel 1/Key 19
//     PlcTask Inputs/GVL_iXlinker.EtherCAT_Master_BKCUCX.TcTerminals210_EK1100_1.TcTerminals210_1BK1250.A_0013_CPx9xx_28_LEDs_Buttons.Channel_1.Key_20 <-> Channel 1/Key 20
//     PlcTask Inputs/GVL_iXlinker.EtherCAT_Master_BKCUCX.TcTerminals210_EK1100_1.TcTerminals210_1BK1250.A_0013_CPx9xx_28_LEDs_Buttons.Channel_1.Key_21 <-> Channel 1/Key 21
//     PlcTask Inputs/GVL_iXlinker.EtherCAT_Master_BKCUCX.TcTerminals210_EK1100_1.TcTerminals210_1BK1250.A_0013_CPx9xx_28_LEDs_Buttons.Channel_1.Key_22 <-> Channel 1/Key 22
//     PlcTask Inputs/GVL_iXlinker.EtherCAT_Master_BKCUCX.TcTerminals210_EK1100_1.TcTerminals210_1BK1250.A_0013_CPx9xx_28_LEDs_Buttons.Channel_1.Key_23 <-> Channel 1/Key 23
//     PlcTask Inputs/GVL_iXlinker.EtherCAT_Master_BKCUCX.TcTerminals210_EK1100_1.TcTerminals210_1BK1250.A_0013_CPx9xx_28_LEDs_Buttons.Channel_1.Key_24 <-> Channel 1/Key 24
//     PlcTask Inputs/GVL_iXlinker.EtherCAT_Master_BKCUCX.TcTerminals210_EK1100_1.TcTerminals210_1BK1250.A_0013_CPx9xx_28_LEDs_Buttons.Channel_1.Key_25 <-> Channel 1/Key 25
//     PlcTask Inputs/GVL_iXlinker.EtherCAT_Master_BKCUCX.TcTerminals210_EK1100_1.TcTerminals210_1BK1250.A_0013_CPx9xx_28_LEDs_Buttons.Channel_1.Key_26 <-> Channel 1/Key 26
//     PlcTask Inputs/GVL_iXlinker.EtherCAT_Master_BKCUCX.TcTerminals210_EK1100_1.TcTerminals210_1BK1250.A_0013_CPx9xx_28_LEDs_Buttons.Channel_1.Key_27 <-> Channel 1/Key 27
//     PlcTask Inputs/GVL_iXlinker.EtherCAT_Master_BKCUCX.TcTerminals210_EK1100_1.TcTerminals210_1BK1250.A_0013_CPx9xx_28_LEDs_Buttons.Channel_1.Key_28 <-> Channel 1/Key 28
//     PlcTask Outputs/GVL_iXlinker.EtherCAT_Master_BKCUCX.TcTerminals210_EK1100_1.TcTerminals210_1BK1250.A_0013_CPx9xx_28_LEDs_Buttons.Channel_1.LED_1 <-> Channel 1/LED 1
//     PlcTask Outputs/GVL_iXlinker.EtherCAT_Master_BKCUCX.TcTerminals210_EK1100_1.TcTerminals210_1BK1250.A_0013_CPx9xx_28_LEDs_Buttons.Channel_1.LED_2 <-> Channel 1/LED 2
//     PlcTask Outputs/GVL_iXlinker.EtherCAT_Master_BKCUCX.TcTerminals210_EK1100_1.TcTerminals210_1BK1250.A_0013_CPx9xx_28_LEDs_Buttons.Channel_1.LED_3 <-> Channel 1/LED 3
//     PlcTask Outputs/GVL_iXlinker.EtherCAT_Master_BKCUCX.TcTerminals210_EK1100_1.TcTerminals210_1BK1250.A_0013_CPx9xx_28_LEDs_Buttons.Channel_1.LED_4 <-> Channel 1/LED 4
//     PlcTask Outputs/GVL_iXlinker.EtherCAT_Master_BKCUCX.TcTerminals210_EK1100_1.TcTerminals210_1BK1250.A_0013_CPx9xx_28_LEDs_Buttons.Channel_1.LED_5 <-> Channel 1/LED 5
//     PlcTask Outputs/GVL_iXlinker.EtherCAT_Master_BKCUCX.TcTerminals210_EK1100_1.TcTerminals210_1BK1250.A_0013_CPx9xx_28_LEDs_Buttons.Channel_1.LED_6 <-> Channel 1/LED 6
//     PlcTask Outputs/GVL_iXlinker.EtherCAT_Master_BKCUCX.TcTerminals210_EK1100_1.TcTerminals210_1BK1250.A_0013_CPx9xx_28_LEDs_Buttons.Channel_1.LED_7 <-> Channel 1/LED 7
//     PlcTask Outputs/GVL_iXlinker.EtherCAT_Master_BKCUCX.TcTerminals210_EK1100_1.TcTerminals210_1BK1250.A_0013_CPx9xx_28_LEDs_Buttons.Channel_1.LED_8 <-> Channel 1/LED 8
//     PlcTask Outputs/GVL_iXlinker.EtherCAT_Master_BKCUCX.TcTerminals210_EK1100_1.TcTerminals210_1BK1250.A_0013_CPx9xx_28_LEDs_Buttons.Channel_1.LED_9 <-> Channel 1/LED 9
//     PlcTask Outputs/GVL_iXlinker.EtherCAT_Master_BKCUCX.TcTerminals210_EK1100_1.TcTerminals210_1BK1250.A_0013_CPx9xx_28_LEDs_Buttons.Channel_1.LED_10 <-> Channel 1/LED 10
//     PlcTask Outputs/GVL_iXlinker.EtherCAT_Master_BKCUCX.TcTerminals210_EK1100_1.TcTerminals210_1BK1250.A_0013_CPx9xx_28_LEDs_Buttons.Channel_1.LED_11 <-> Channel 1/LED 11
//     PlcTask Outputs/GVL_iXlinker.EtherCAT_Master_BKCUCX.TcTerminals210_EK1100_1.TcTerminals210_1BK1250.A_0013_CPx9xx_28_LEDs_Buttons.Channel_1.LED_12 <-> Channel 1/LED 12
//     PlcTask Outputs/GVL_iXlinker.EtherCAT_Master_BKCUCX.TcTerminals210_EK1100_1.TcTerminals210_1BK1250.A_0013_CPx9xx_28_LEDs_Buttons.Channel_1.LED_13 <-> Channel 1/LED 13
//     PlcTask Outputs/GVL_iXlinker.EtherCAT_Master_BKCUCX.TcTerminals210_EK1100_1.TcTerminals210_1BK1250.A_0013_CPx9xx_28_LEDs_Buttons.Channel_1.LED_14 <-> Channel 1/LED 14
//     PlcTask Outputs/GVL_iXlinker.EtherCAT_Master_BKCUCX.TcTerminals210_EK1100_1.TcTerminals210_1BK1250.A_0013_CPx9xx_28_LEDs_Buttons.Channel_1.LED_15 <-> Channel 1/LED 15
//     PlcTask Outputs/GVL_iXlinker.EtherCAT_Master_BKCUCX.TcTerminals210_EK1100_1.TcTerminals210_1BK1250.A_0013_CPx9xx_28_LEDs_Buttons.Channel_1.LED_16 <-> Channel 1/LED 16
//     PlcTask Outputs/GVL_iXlinker.EtherCAT_Master_BKCUCX.TcTerminals210_EK1100_1.TcTerminals210_1BK1250.A_0013_CPx9xx_28_LEDs_Buttons.Channel_1.LED_17 <-> Channel 1/LED 17
//     PlcTask Outputs/GVL_iXlinker.EtherCAT_Master_BKCUCX.TcTerminals210_EK1100_1.TcTerminals210_1BK1250.A_0013_CPx9xx_28_LEDs_Buttons.Channel_1.LED_18 <-> Channel 1/LED 18
//     PlcTask Outputs/GVL_iXlinker.EtherCAT_Master_BKCUCX.TcTerminals210_EK1100_1.TcTerminals210_1BK1250.A_0013_CPx9xx_28_LEDs_Buttons.Channel_1.LED_19 <-> Channel 1/LED 19
//     PlcTask Outputs/GVL_iXlinker.EtherCAT_Master_BKCUCX.TcTerminals210_EK1100_1.TcTerminals210_1BK1250.A_0013_CPx9xx_28_LEDs_Buttons.Channel_1.LED_20 <-> Channel 1/LED 20
//     PlcTask Outputs/GVL_iXlinker.EtherCAT_Master_BKCUCX.TcTerminals210_EK1100_1.TcTerminals210_1BK1250.A_0013_CPx9xx_28_LEDs_Buttons.Channel_1.LED_21 <-> Channel 1/LED 21
//     PlcTask Outputs/GVL_iXlinker.EtherCAT_Master_BKCUCX.TcTerminals210_EK1100_1.TcTerminals210_1BK1250.A_0013_CPx9xx_28_LEDs_Buttons.Channel_1.LED_22 <-> Channel 1/LED 22
//     PlcTask Outputs/GVL_iXlinker.EtherCAT_Master_BKCUCX.TcTerminals210_EK1100_1.TcTerminals210_1BK1250.A_0013_CPx9xx_28_LEDs_Buttons.Channel_1.LED_23 <-> Channel 1/LED 23
//     PlcTask Outputs/GVL_iXlinker.EtherCAT_Master_BKCUCX.TcTerminals210_EK1100_1.TcTerminals210_1BK1250.A_0013_CPx9xx_28_LEDs_Buttons.Channel_1.LED_24 <-> Channel 1/LED 24
//     PlcTask Outputs/GVL_iXlinker.EtherCAT_Master_BKCUCX.TcTerminals210_EK1100_1.TcTerminals210_1BK1250.A_0013_CPx9xx_28_LEDs_Buttons.Channel_1.LED_25 <-> Channel 1/LED 25
//     PlcTask Outputs/GVL_iXlinker.EtherCAT_Master_BKCUCX.TcTerminals210_EK1100_1.TcTerminals210_1BK1250.A_0013_CPx9xx_28_LEDs_Buttons.Channel_1.LED_26 <-> Channel 1/LED 26
//     PlcTask Outputs/GVL_iXlinker.EtherCAT_Master_BKCUCX.TcTerminals210_EK1100_1.TcTerminals210_1BK1250.A_0013_CPx9xx_28_LEDs_Buttons.Channel_1.LED_27 <-> Channel 1/LED 27
//     PlcTask Outputs/GVL_iXlinker.EtherCAT_Master_BKCUCX.TcTerminals210_EK1100_1.TcTerminals210_1BK1250.A_0013_CPx9xx_28_LEDs_Buttons.Channel_1.LED_28 <-> Channel 1/LED 28
//   PLC/PLC Instance <-> EtherCAT Master BKCUCX/TcTerminals210_EK1100_1/TcTerminals210_1BK1250/A_0015(CPx9xx-3-2 LEDs/Buttons/Inputs)
//     PlcTask Inputs/GVL_iXlinker.EtherCAT_Master_BKCUCX.TcTerminals210_EK1100_1.TcTerminals210_1BK1250.A_0015_CPx9xx_3_2_LEDs_Buttons_Inputs.Channel_1.Key_1 <-> Channel 1/Key 1
//     PlcTask Inputs/GVL_iXlinker.EtherCAT_Master_BKCUCX.TcTerminals210_EK1100_1.TcTerminals210_1BK1250.A_0015_CPx9xx_3_2_LEDs_Buttons_Inputs.Channel_1.Key_2 <-> Channel 1/Key 2
//     PlcTask Inputs/GVL_iXlinker.EtherCAT_Master_BKCUCX.TcTerminals210_EK1100_1.TcTerminals210_1BK1250.A_0015_CPx9xx_3_2_LEDs_Buttons_Inputs.Channel_1.Key_3 <-> Channel 1/Key 3
//     PlcTask Inputs/GVL_iXlinker.EtherCAT_Master_BKCUCX.TcTerminals210_EK1100_1.TcTerminals210_1BK1250.A_0015_CPx9xx_3_2_LEDs_Buttons_Inputs.Channel_1.Input_1 <-> Channel 1/Input 1
//     PlcTask Inputs/GVL_iXlinker.EtherCAT_Master_BKCUCX.TcTerminals210_EK1100_1.TcTerminals210_1BK1250.A_0015_CPx9xx_3_2_LEDs_Buttons_Inputs.Channel_1.Input_2 <-> Channel 1/Input 2
//     PlcTask Inputs/GVL_iXlinker.EtherCAT_Master_BKCUCX.TcTerminals210_EK1100_1.TcTerminals210_1BK1250.A_0015_CPx9xx_3_2_LEDs_Buttons_Inputs.Channel_1.Input_3 <-> Channel 1/Input 3
//     PlcTask Outputs/GVL_iXlinker.EtherCAT_Master_BKCUCX.TcTerminals210_EK1100_1.TcTerminals210_1BK1250.A_0015_CPx9xx_3_2_LEDs_Buttons_Inputs.Channel_1.LED_1 <-> Channel 1/LED 1
//     PlcTask Outputs/GVL_iXlinker.EtherCAT_Master_BKCUCX.TcTerminals210_EK1100_1.TcTerminals210_1BK1250.A_0015_CPx9xx_3_2_LEDs_Buttons_Inputs.Channel_1.LED_2 <-> Channel 1/LED 2
//     PlcTask Outputs/GVL_iXlinker.EtherCAT_Master_BKCUCX.TcTerminals210_EK1100_1.TcTerminals210_1BK1250.A_0015_CPx9xx_3_2_LEDs_Buttons_Inputs.Channel_1.LED_3 <-> Channel 1/LED 3
//   PLC/PLC Instance <-> EtherCAT Master BKCUCX/TcTerminals210_EK1100_1/TcTerminals210_1BK1250/A_0016(CPx9xx-4-2 LEDs/Buttons/Inputs)
//     PlcTask Inputs/GVL_iXlinker.EtherCAT_Master_BKCUCX.TcTerminals210_EK1100_1.TcTerminals210_1BK1250.A_0016_CPx9xx_4_2_LEDs_Buttons_Inputs.Channel_1.Key_1 <-> Channel 1/Key 1
//     PlcTask Inputs/GVL_iXlinker.EtherCAT_Master_BKCUCX.TcTerminals210_EK1100_1.TcTerminals210_1BK1250.A_0016_CPx9xx_4_2_LEDs_Buttons_Inputs.Channel_1.Key_2 <-> Channel 1/Key 2
//     PlcTask Inputs/GVL_iXlinker.EtherCAT_Master_BKCUCX.TcTerminals210_EK1100_1.TcTerminals210_1BK1250.A_0016_CPx9xx_4_2_LEDs_Buttons_Inputs.Channel_1.Key_3 <-> Channel 1/Key 3
//     PlcTask Inputs/GVL_iXlinker.EtherCAT_Master_BKCUCX.TcTerminals210_EK1100_1.TcTerminals210_1BK1250.A_0016_CPx9xx_4_2_LEDs_Buttons_Inputs.Channel_1.Key_4 <-> Channel 1/Key 4
//     PlcTask Inputs/GVL_iXlinker.EtherCAT_Master_BKCUCX.TcTerminals210_EK1100_1.TcTerminals210_1BK1250.A_0016_CPx9xx_4_2_LEDs_Buttons_Inputs.Channel_1.Input_1 <-> Channel 1/Input 1
//     PlcTask Inputs/GVL_iXlinker.EtherCAT_Master_BKCUCX.TcTerminals210_EK1100_1.TcTerminals210_1BK1250.A_0016_CPx9xx_4_2_LEDs_Buttons_Inputs.Channel_1.Input_2 <-> Channel 1/Input 2
//     PlcTask Inputs/GVL_iXlinker.EtherCAT_Master_BKCUCX.TcTerminals210_EK1100_1.TcTerminals210_1BK1250.A_0016_CPx9xx_4_2_LEDs_Buttons_Inputs.Channel_1.Input_3 <-> Channel 1/Input 3
//     PlcTask Inputs/GVL_iXlinker.EtherCAT_Master_BKCUCX.TcTerminals210_EK1100_1.TcTerminals210_1BK1250.A_0016_CPx9xx_4_2_LEDs_Buttons_Inputs.Channel_1.Input_4 <-> Channel 1/Input 4
//     PlcTask Outputs/GVL_iXlinker.EtherCAT_Master_BKCUCX.TcTerminals210_EK1100_1.TcTerminals210_1BK1250.A_0016_CPx9xx_4_2_LEDs_Buttons_Inputs.Channel_1.LED_1 <-> Channel 1/LED 1
//     PlcTask Outputs/GVL_iXlinker.EtherCAT_Master_BKCUCX.TcTerminals210_EK1100_1.TcTerminals210_1BK1250.A_0016_CPx9xx_4_2_LEDs_Buttons_Inputs.Channel_1.LED_2 <-> Channel 1/LED 2
//     PlcTask Outputs/GVL_iXlinker.EtherCAT_Master_BKCUCX.TcTerminals210_EK1100_1.TcTerminals210_1BK1250.A_0016_CPx9xx_4_2_LEDs_Buttons_Inputs.Channel_1.LED_3 <-> Channel 1/LED 3
//     PlcTask Outputs/GVL_iXlinker.EtherCAT_Master_BKCUCX.TcTerminals210_EK1100_1.TcTerminals210_1BK1250.A_0016_CPx9xx_4_2_LEDs_Buttons_Inputs.Channel_1.LED_4 <-> Channel 1/LED 4
//   PLC/PLC Instance <-> EtherCAT Master BKCUCX/TcTerminals210_EK1100_1/TcTerminals210_1BK1250/A_0129(KL 1002, 2 Ch. Input (24V, 3.0ms))
//     PlcTask Inputs/GVL_iXlinker.EtherCAT_Master_BKCUCX.TcTerminals210_EK1100_1.TcTerminals210_1BK1250.A_0129_KL_1002_2_Ch_Input_24V_3_0ms.Channel_1.Input <-> Channel 1/Input
//     PlcTask Inputs/GVL_iXlinker.EtherCAT_Master_BKCUCX.TcTerminals210_EK1100_1.TcTerminals210_1BK1250.A_0129_KL_1002_2_Ch_Input_24V_3_0ms.Channel_2.Input <-> Channel 2/Input
//   PLC/PLC Instance <-> EtherCAT Master BKCUCX/TcTerminals210_EK1100_1/TcTerminals210_1BK1250/A_0130(CPx9xx-E-Stop)
//     PlcTask Inputs/GVL_iXlinker.EtherCAT_Master_BKCUCX.TcTerminals210_EK1100_1.TcTerminals210_1BK1250.A_0130_CPx9xx_E_Stop.Channel_1.E_Stop <-> Channel 1/E-Stop
//   PLC/PLC Instance <-> EtherCAT Master BKCUCX/TcTerminals210_EK1100_1/TcTerminals210_1BK1250/A_0131(KL 1012, 2 Ch. Input (24V, 0.2ms))
//     PlcTask Inputs/GVL_iXlinker.EtherCAT_Master_BKCUCX.TcTerminals210_EK1100_1.TcTerminals210_1BK1250.A_0131_KL_1012_2_Ch_Input_24V_0_2ms.Channel_1.Input <-> Channel 1/Input
//     PlcTask Inputs/GVL_iXlinker.EtherCAT_Master_BKCUCX.TcTerminals210_EK1100_1.TcTerminals210_1BK1250.A_0131_KL_1012_2_Ch_Input_24V_0_2ms.Channel_2.Input <-> Channel 2/Input
//   PLC/PLC Instance <-> EtherCAT Master BKCUCX/TcTerminals210_EK1100_1/TcTerminals210_1BK1250/A_0132(KL 1032, 2 Ch. Input (48V, 3.0ms))
